(* Schneider Machine Expert - Basic project control_2, file version 2.9.0.0 *)
(* ProjectInformations: Name=Nuevo proyecto *)

HARDWARE
  Cpu 0: TM221M16R/G
  EthernetConfiguration: NetworkName=M221, IpAllocationMode=FixedAddress, IpAddress=0.0.0.0, SubnetMask=0.0.0.0
  SerialLineConfiguration: Baud=Baud19200, Parity=ParityEven, DataBits=DataBits8, StopBits=StopBits1, PhysicalMedium=PhysicalMediumRs485, TransmissionMode=TransmissionModeModbusRtu, SlaveId=1, Addressing=SlaveAddressing
  MastTask: UsePeriodScanMode=true, PeriodScan=50
  FastTask: Period=255
  CpuBehavior: StartingMode=StartAsPreviousState, AutoSaveRamOnEeprom=true, WatchdogPeriod=250

SYMBOLS  (address, symbol, comment, settings)
  %MW271    CONT
  %MW500    ERR
  %MW501    VEL
  %MW502    THETA
  %MW503    CRISP
  %MF1      REAL_ERROR
  %MF10     ENL
  %MF19     ENM
  %MF28     ENP
  %MF37     EZ
  %MF46     EPP
  %MF55     EPM
  %MF64     EPL
  %MF67     REAL_VEL
  %MF76     VNL
  %MF85     VNM
  %MF94     VNP
  %MF103    VZ
  %MF112    VPP
  %MF121    VPM
  %MF130    VPL
  %MF133    REAL_THETA
  %MF142    NL
  %MF151    NM
  %MF160    Z
  %MF169    PM
  %MF178    PL
  %MF181    W1
  %MF184    W2
  %MF187    W3
  %MF190    W4
  %MF193    W5
  %MF196    W6
  %MF199    W7
  %MF202    W8
  %MF205    W9
  %MF208    W10
  %MF211    W11
  %MF214    W12
  %MF217    W13
  %MF220    W14
  %MF223    W15
  %MF226    W16
  %MF229    W17
  %MF232    W18
  %MF235    W19
  %MF238    W20
  %MF241    W21
  %MF244    W22
  %MF247    W23
  %MF250    W24
  %MF253    W25
  %MF256    U_NL
  %MF259    U_NM
  %MF262    U_ZR
  %MF265    U_PM
  %MF268    U_PL
  %KF1      F_CONV  [Value=1000]
  %KF4      CONV_OUTPUT  [Value=100]

POU Nuevo POU
  (* SectionNumber=1 *)

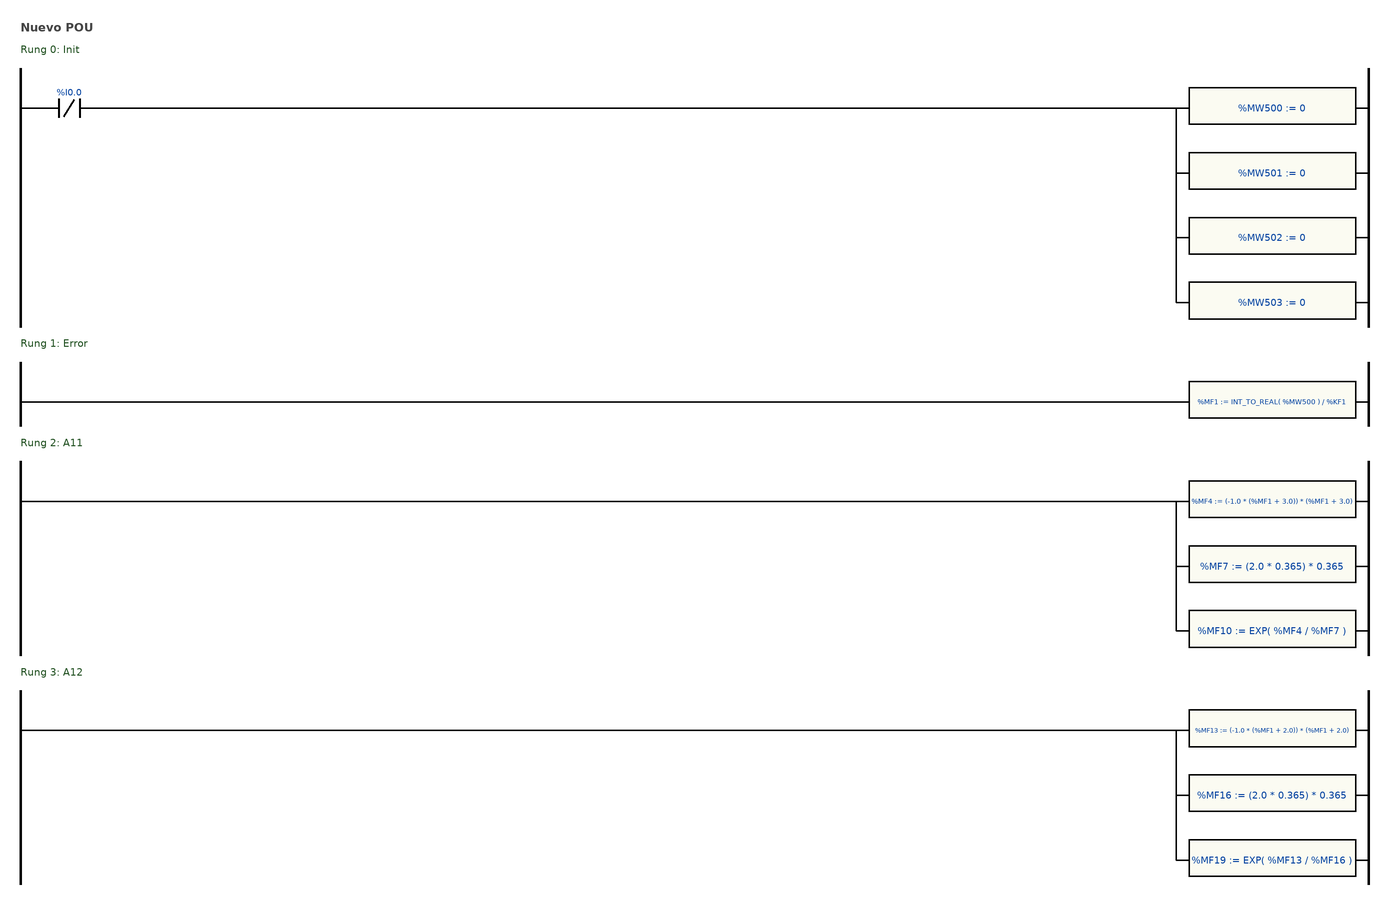

// Rung 0: Init
  LDN %I0.0
  [ %MW500 := 0 ]         (* ERR *)
  [ %MW501 := 0 ]         (* VEL *)
  [ %MW502 := 0 ]         (* THETA *)
  [ %MW503 := 0 ]         (* CRISP *)
  // as ST:
  //   IF NOT %I0.0 THEN ERR := 0; END_IF;
  //   IF NOT %I0.0 THEN VEL := 0; END_IF;
  //   IF NOT %I0.0 THEN THETA := 0; END_IF;
  //   IF NOT %I0.0 THEN CRISP := 0; END_IF;

// Rung 1: Error
  LD 1
  [ %MF1 := INT_TO_REAL ( %MW500 ) / %KF1 ](* REAL_ERROR, ERR, F_CONV *)
  // as ST:
  //   REAL_ERROR := INT_TO_REAL ( ERR ) / F_CONV;

// Rung 2: A11
  LD 1
  [ %MF4 := ( -1.0 * ( %MF1 + 3.0 ) ) * ( %MF1 + 3.0 ) ](* REAL_ERROR, REAL_ERROR *)
  [ %MF7 := ( 2.0 * 0.365 ) * 0.365 ]
  [ %MF10 := EXP ( %MF4 / %MF7 ) ](* ENL *)
  // as ST:
  //   %MF4 := ( -1.0 * ( REAL_ERROR + 3.0 ) ) * ( REAL_ERROR + 3.0 );
  //   %MF7 := ( 2.0 * 0.365 ) * 0.365;
  //   ENL := EXP ( %MF4 / %MF7 );

// Rung 3: A12
  LD 1
  [ %MF13 := ( -1.0 * ( %MF1 + 2.0 ) ) * ( %MF1 + 2.0 ) ](* REAL_ERROR, REAL_ERROR *)
  [ %MF16 := ( 2.0 * 0.365 ) * 0.365 ]
  [ %MF19 := EXP ( %MF13 / %MF16 ) ](* ENM *)
  // as ST:
  //   %MF13 := ( -1.0 * ( REAL_ERROR + 2.0 ) ) * ( REAL_ERROR + 2.0 );
  //   %MF16 := ( 2.0 * 0.365 ) * 0.365;
  //   ENM := EXP ( %MF13 / %MF16 );

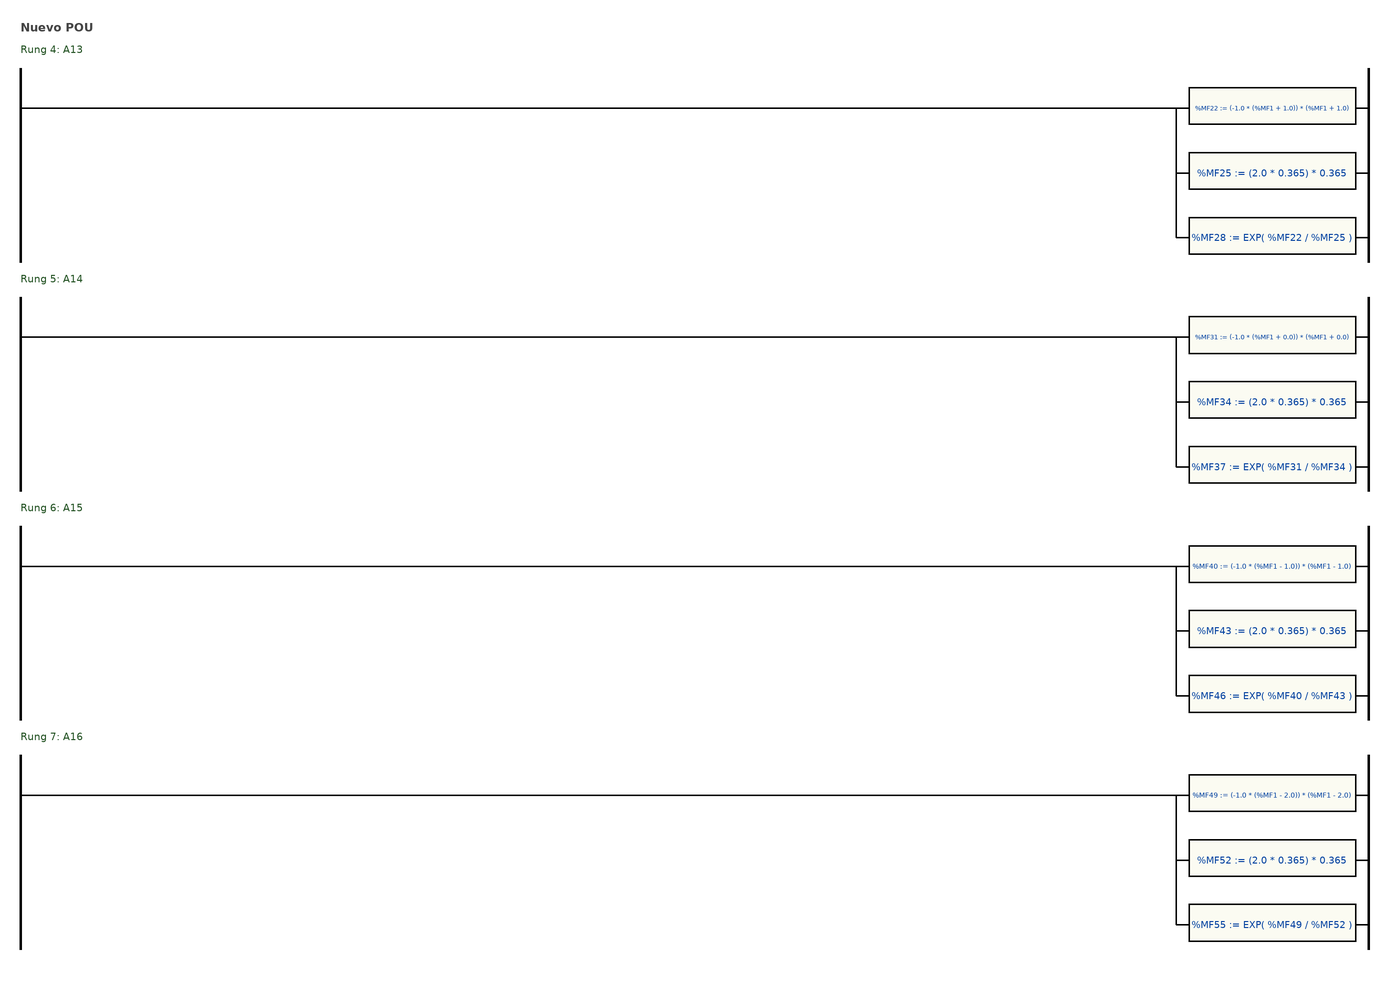

// Rung 4: A13
  LD 1
  [ %MF22 := ( -1.0 * ( %MF1 + 1.0 ) ) * ( %MF1 + 1.0 ) ](* REAL_ERROR, REAL_ERROR *)
  [ %MF25 := ( 2.0 * 0.365 ) * 0.365 ]
  [ %MF28 := EXP ( %MF22 / %MF25 ) ](* ENP *)
  // as ST:
  //   %MF22 := ( -1.0 * ( REAL_ERROR + 1.0 ) ) * ( REAL_ERROR + 1.0 );
  //   %MF25 := ( 2.0 * 0.365 ) * 0.365;
  //   ENP := EXP ( %MF22 / %MF25 );

// Rung 5: A14
  LD 1
  [ %MF31 := ( -1.0 * ( %MF1 + 0.0 ) ) * ( %MF1 + 0.0 ) ](* REAL_ERROR, REAL_ERROR *)
  [ %MF34 := ( 2.0 * 0.365 ) * 0.365 ]
  [ %MF37 := EXP ( %MF31 / %MF34 ) ](* EZ *)
  // as ST:
  //   %MF31 := ( -1.0 * ( REAL_ERROR + 0.0 ) ) * ( REAL_ERROR + 0.0 );
  //   %MF34 := ( 2.0 * 0.365 ) * 0.365;
  //   EZ := EXP ( %MF31 / %MF34 );

// Rung 6: A15
  LD 1
  [ %MF40 := ( -1.0 * ( %MF1 - 1.0 ) ) * ( %MF1 - 1.0 ) ](* REAL_ERROR, REAL_ERROR *)
  [ %MF43 := ( 2.0 * 0.365 ) * 0.365 ]
  [ %MF46 := EXP ( %MF40 / %MF43 ) ](* EPP *)
  // as ST:
  //   %MF40 := ( -1.0 * ( REAL_ERROR - 1.0 ) ) * ( REAL_ERROR - 1.0 );
  //   %MF43 := ( 2.0 * 0.365 ) * 0.365;
  //   EPP := EXP ( %MF40 / %MF43 );

// Rung 7: A16
  LD 1
  [ %MF49 := ( -1.0 * ( %MF1 - 2.0 ) ) * ( %MF1 - 2.0 ) ](* REAL_ERROR, REAL_ERROR *)
  [ %MF52 := ( 2.0 * 0.365 ) * 0.365 ]
  [ %MF55 := EXP ( %MF49 / %MF52 ) ](* EPM *)
  // as ST:
  //   %MF49 := ( -1.0 * ( REAL_ERROR - 2.0 ) ) * ( REAL_ERROR - 2.0 );
  //   %MF52 := ( 2.0 * 0.365 ) * 0.365;
  //   EPM := EXP ( %MF49 / %MF52 );

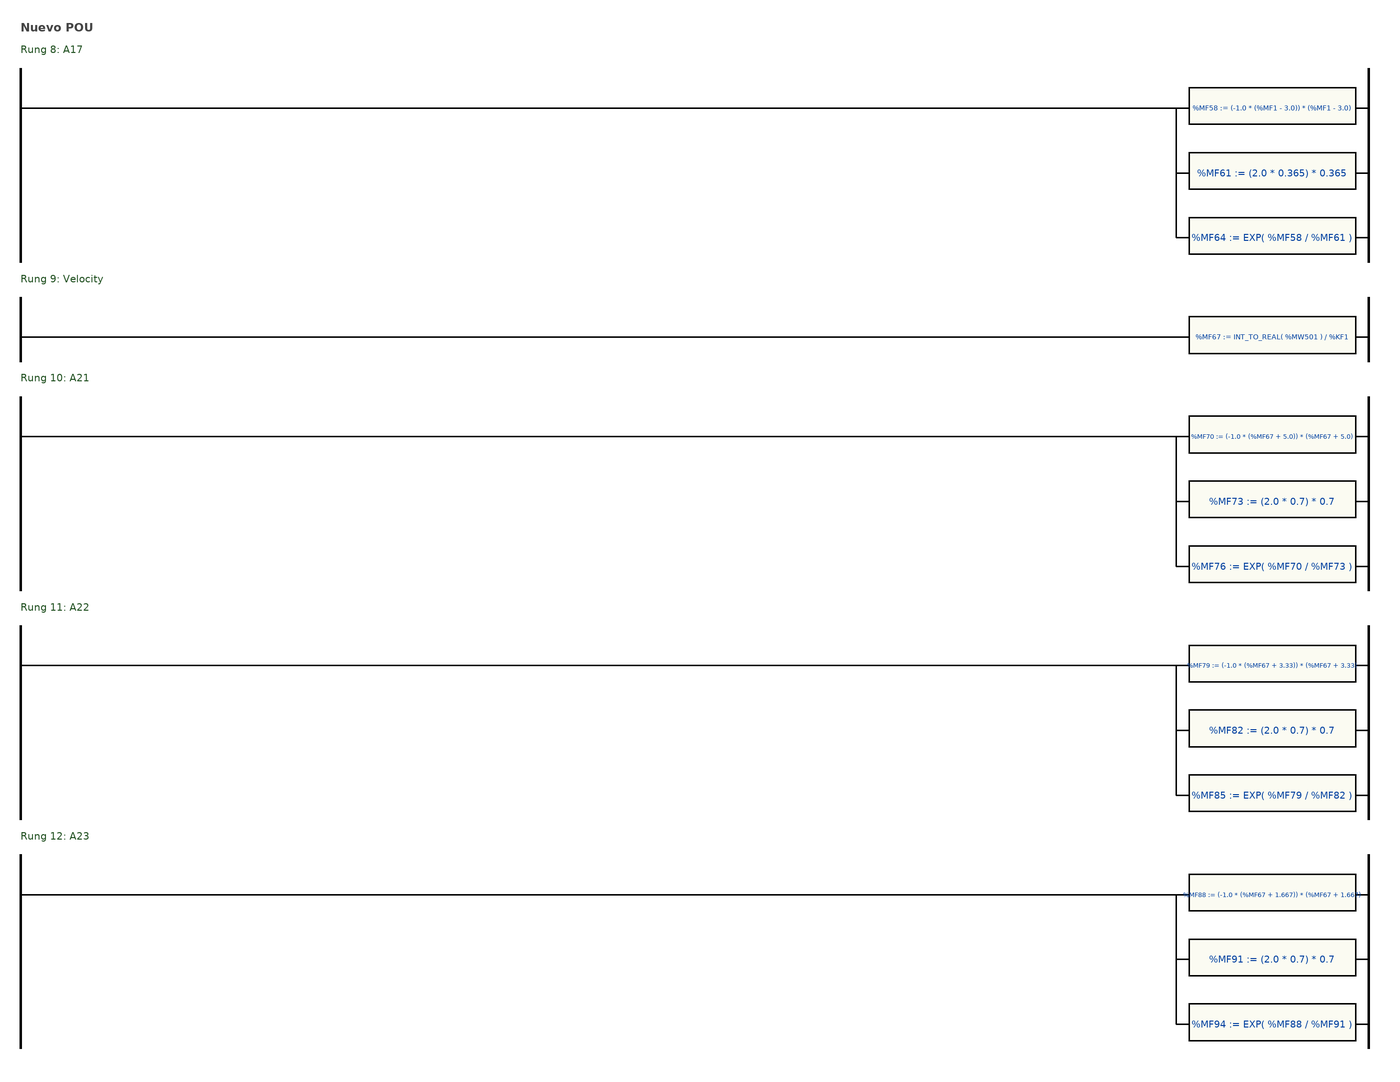

// Rung 8: A17
  LD 1
  [ %MF58 := ( -1.0 * ( %MF1 - 3.0 ) ) * ( %MF1 - 3.0 ) ](* REAL_ERROR, REAL_ERROR *)
  [ %MF61 := ( 2.0 * 0.365 ) * 0.365 ]
  [ %MF64 := EXP ( %MF58 / %MF61 ) ](* EPL *)
  // as ST:
  //   %MF58 := ( -1.0 * ( REAL_ERROR - 3.0 ) ) * ( REAL_ERROR - 3.0 );
  //   %MF61 := ( 2.0 * 0.365 ) * 0.365;
  //   EPL := EXP ( %MF58 / %MF61 );

// Rung 9: Velocity
  LD 1
  [ %MF67 := INT_TO_REAL ( %MW501 ) / %KF1 ](* REAL_VEL, VEL, F_CONV *)
  // as ST:
  //   REAL_VEL := INT_TO_REAL ( VEL ) / F_CONV;

// Rung 10: A21
  LD 1
  [ %MF70 := ( -1.0 * ( %MF67 + 5.0 ) ) * ( %MF67 + 5.0 ) ](* REAL_VEL, REAL_VEL *)
  [ %MF73 := ( 2.0 * 0.7 ) * 0.7 ]
  [ %MF76 := EXP ( %MF70 / %MF73 ) ](* VNL *)
  // as ST:
  //   %MF70 := ( -1.0 * ( REAL_VEL + 5.0 ) ) * ( REAL_VEL + 5.0 );
  //   %MF73 := ( 2.0 * 0.7 ) * 0.7;
  //   VNL := EXP ( %MF70 / %MF73 );

// Rung 11: A22
  LD 1
  [ %MF79 := ( -1.0 * ( %MF67 + 3.33 ) ) * ( %MF67 + 3.33 ) ](* REAL_VEL, REAL_VEL *)
  [ %MF82 := ( 2.0 * 0.7 ) * 0.7 ]
  [ %MF85 := EXP ( %MF79 / %MF82 ) ](* VNM *)
  // as ST:
  //   %MF79 := ( -1.0 * ( REAL_VEL + 3.33 ) ) * ( REAL_VEL + 3.33 );
  //   %MF82 := ( 2.0 * 0.7 ) * 0.7;
  //   VNM := EXP ( %MF79 / %MF82 );

// Rung 12: A23
  LD 1
  [ %MF88 := ( -1.0 * ( %MF67 + 1.667 ) ) * ( %MF67 + 1.667 ) ](* REAL_VEL, REAL_VEL *)
  [ %MF91 := ( 2.0 * 0.7 ) * 0.7 ]
  [ %MF94 := EXP ( %MF88 / %MF91 ) ](* VNP *)
  // as ST:
  //   %MF88 := ( -1.0 * ( REAL_VEL + 1.667 ) ) * ( REAL_VEL + 1.667 );
  //   %MF91 := ( 2.0 * 0.7 ) * 0.7;
  //   VNP := EXP ( %MF88 / %MF91 );

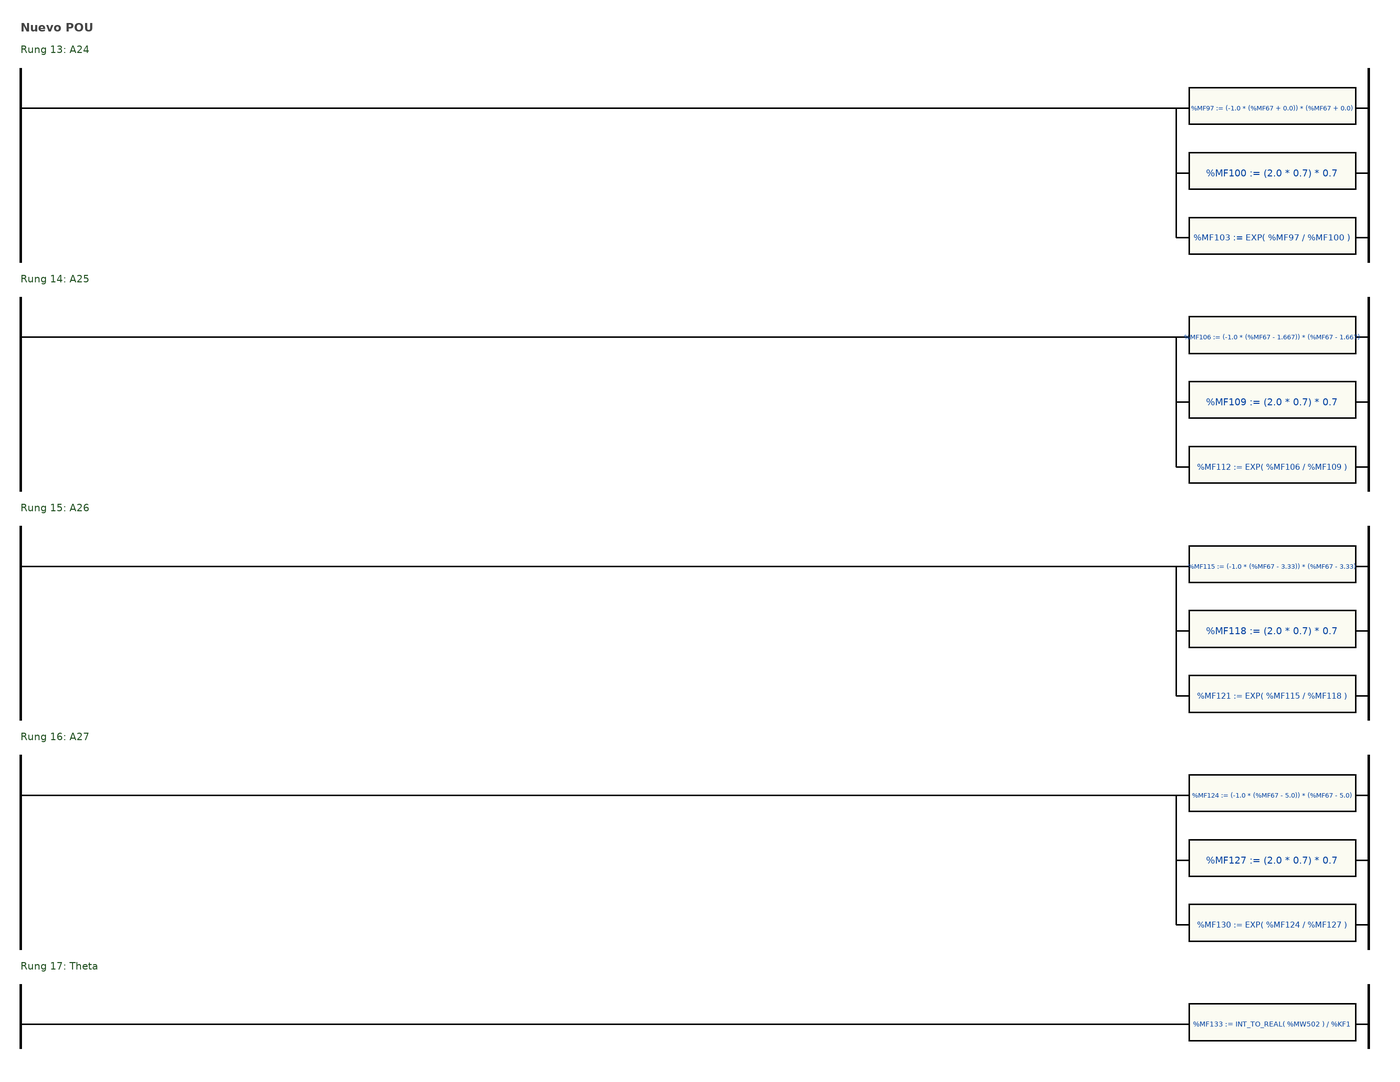

// Rung 13: A24
  LD 1
  [ %MF97 := ( -1.0 * ( %MF67 + 0.0 ) ) * ( %MF67 + 0.0 ) ](* REAL_VEL, REAL_VEL *)
  [ %MF100 := ( 2.0 * 0.7 ) * 0.7 ]
  [ %MF103 := EXP ( %MF97 / %MF100 ) ](* VZ *)
  // as ST:
  //   %MF97 := ( -1.0 * ( REAL_VEL + 0.0 ) ) * ( REAL_VEL + 0.0 );
  //   %MF100 := ( 2.0 * 0.7 ) * 0.7;
  //   VZ := EXP ( %MF97 / %MF100 );

// Rung 14: A25
  LD 1
  [ %MF106 := ( -1.0 * ( %MF67 - 1.667 ) ) * ( %MF67 - 1.667 ) ](* REAL_VEL, REAL_VEL *)
  [ %MF109 := ( 2.0 * 0.7 ) * 0.7 ]
  [ %MF112 := EXP ( %MF106 / %MF109 ) ](* VPP *)
  // as ST:
  //   %MF106 := ( -1.0 * ( REAL_VEL - 1.667 ) ) * ( REAL_VEL - 1.667 );
  //   %MF109 := ( 2.0 * 0.7 ) * 0.7;
  //   VPP := EXP ( %MF106 / %MF109 );

// Rung 15: A26
  LD 1
  [ %MF115 := ( -1.0 * ( %MF67 - 3.33 ) ) * ( %MF67 - 3.33 ) ](* REAL_VEL, REAL_VEL *)
  [ %MF118 := ( 2.0 * 0.7 ) * 0.7 ]
  [ %MF121 := EXP ( %MF115 / %MF118 ) ](* VPM *)
  // as ST:
  //   %MF115 := ( -1.0 * ( REAL_VEL - 3.33 ) ) * ( REAL_VEL - 3.33 );
  //   %MF118 := ( 2.0 * 0.7 ) * 0.7;
  //   VPM := EXP ( %MF115 / %MF118 );

// Rung 16: A27
  LD 1
  [ %MF124 := ( -1.0 * ( %MF67 - 5.0 ) ) * ( %MF67 - 5.0 ) ](* REAL_VEL, REAL_VEL *)
  [ %MF127 := ( 2.0 * 0.7 ) * 0.7 ]
  [ %MF130 := EXP ( %MF124 / %MF127 ) ](* VPL *)
  // as ST:
  //   %MF124 := ( -1.0 * ( REAL_VEL - 5.0 ) ) * ( REAL_VEL - 5.0 );
  //   %MF127 := ( 2.0 * 0.7 ) * 0.7;
  //   VPL := EXP ( %MF124 / %MF127 );

// Rung 17: Theta
  LD 1
  [ %MF133 := INT_TO_REAL ( %MW502 ) / %KF1 ](* REAL_THETA, THETA, F_CONV *)
  // as ST:
  //   REAL_THETA := INT_TO_REAL ( THETA ) / F_CONV;

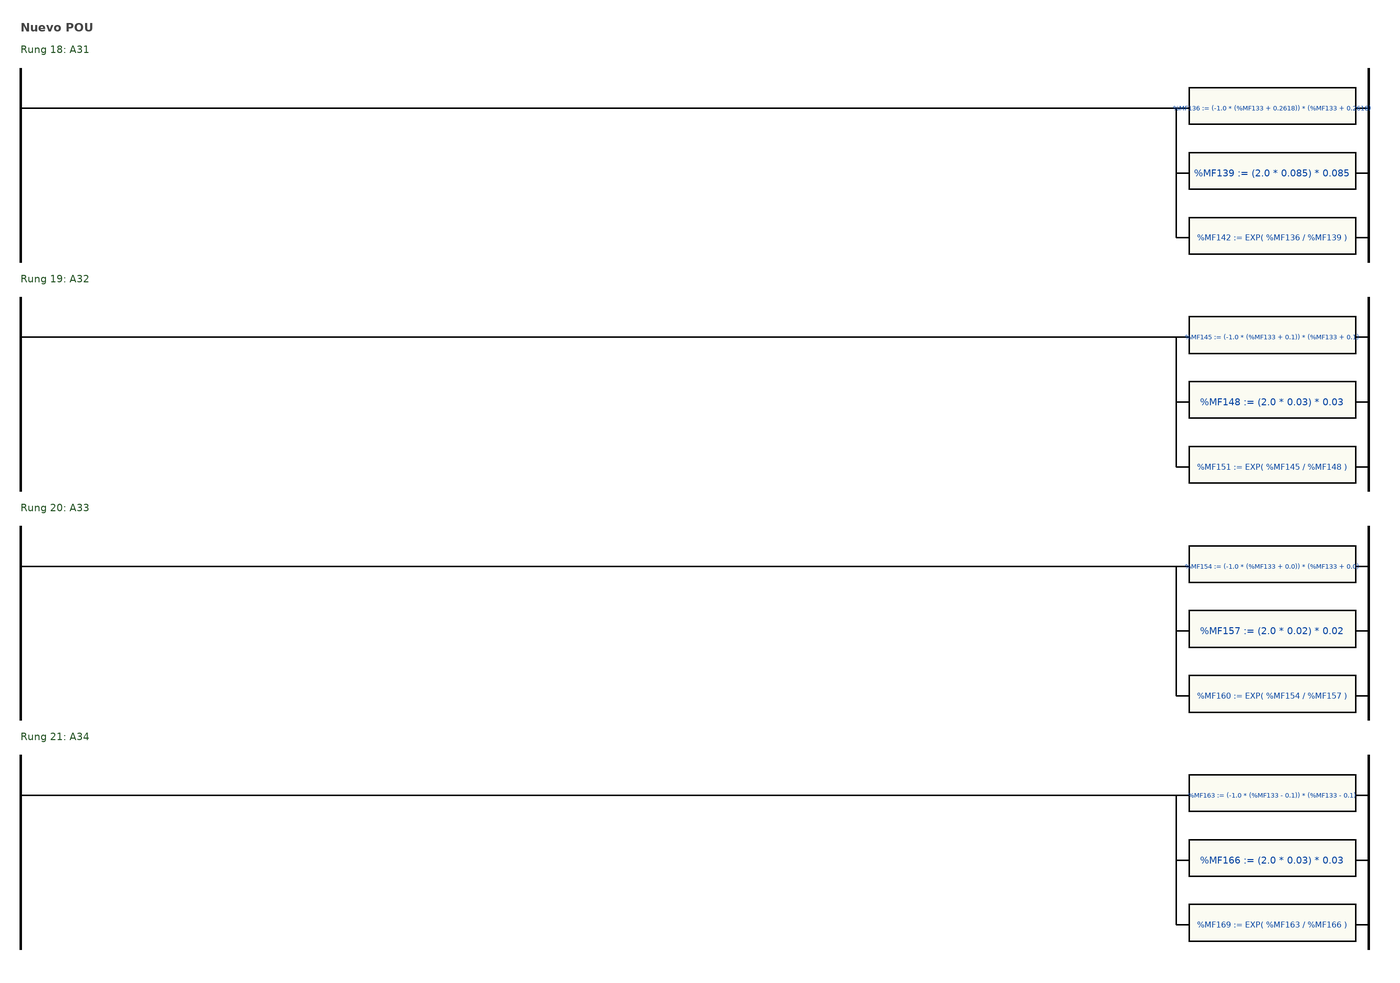

// Rung 18: A31
  LD 1
  [ %MF136 := ( -1.0 * ( %MF133 + 0.2618 ) ) * ( %MF133 + 0.2618 ) ](* REAL_THETA, REAL_THETA *)
  [ %MF139 := ( 2.0 * 0.085 ) * 0.085 ]
  [ %MF142 := EXP ( %MF136 / %MF139 ) ](* NL *)
  // as ST:
  //   %MF136 := ( -1.0 * ( REAL_THETA + 0.2618 ) ) * ( REAL_THETA + 0.2618 );
  //   %MF139 := ( 2.0 * 0.085 ) * 0.085;
  //   NL := EXP ( %MF136 / %MF139 );

// Rung 19: A32
  LD 1
  [ %MF145 := ( -1.0 * ( %MF133 + 0.1 ) ) * ( %MF133 + 0.1 ) ](* REAL_THETA, REAL_THETA *)
  [ %MF148 := ( 2.0 * 0.03 ) * 0.03 ]
  [ %MF151 := EXP ( %MF145 / %MF148 ) ](* NM *)
  // as ST:
  //   %MF145 := ( -1.0 * ( REAL_THETA + 0.1 ) ) * ( REAL_THETA + 0.1 );
  //   %MF148 := ( 2.0 * 0.03 ) * 0.03;
  //   NM := EXP ( %MF145 / %MF148 );

// Rung 20: A33
  LD 1
  [ %MF154 := ( -1.0 * ( %MF133 + 0.0 ) ) * ( %MF133 + 0.0 ) ](* REAL_THETA, REAL_THETA *)
  [ %MF157 := ( 2.0 * 0.02 ) * 0.02 ]
  [ %MF160 := EXP ( %MF154 / %MF157 ) ](* Z *)
  // as ST:
  //   %MF154 := ( -1.0 * ( REAL_THETA + 0.0 ) ) * ( REAL_THETA + 0.0 );
  //   %MF157 := ( 2.0 * 0.02 ) * 0.02;
  //   Z := EXP ( %MF154 / %MF157 );

// Rung 21: A34
  LD 1
  [ %MF163 := ( -1.0 * ( %MF133 - 0.1 ) ) * ( %MF133 - 0.1 ) ](* REAL_THETA, REAL_THETA *)
  [ %MF166 := ( 2.0 * 0.03 ) * 0.03 ]
  [ %MF169 := EXP ( %MF163 / %MF166 ) ](* PM *)
  // as ST:
  //   %MF163 := ( -1.0 * ( REAL_THETA - 0.1 ) ) * ( REAL_THETA - 0.1 );
  //   %MF166 := ( 2.0 * 0.03 ) * 0.03;
  //   PM := EXP ( %MF163 / %MF166 );

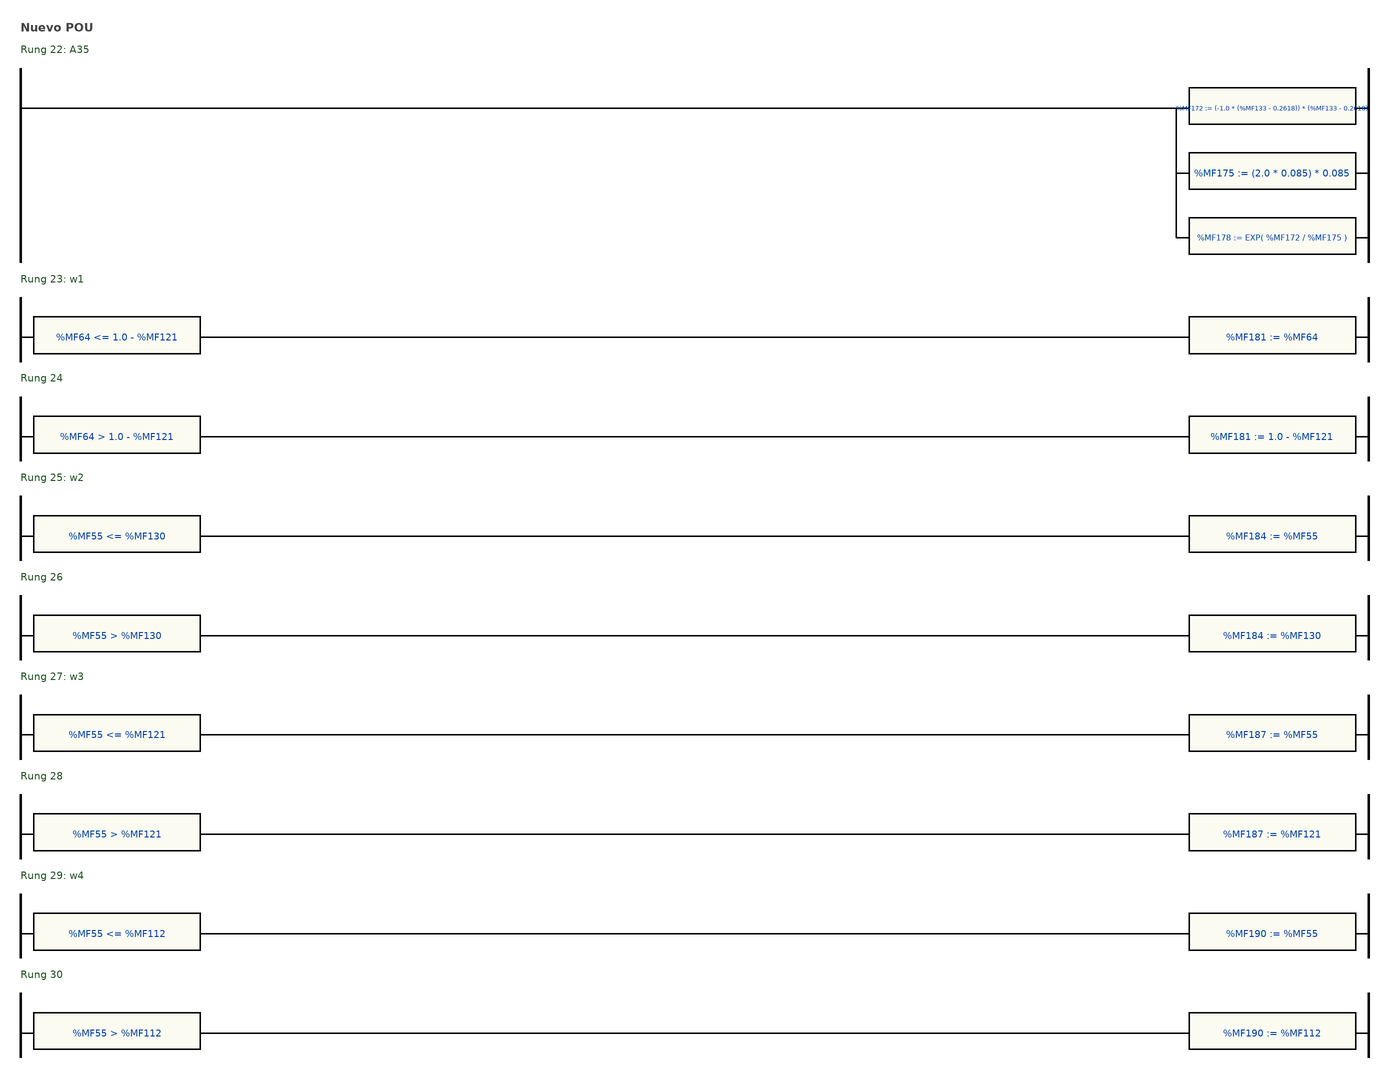

// Rung 22: A35
  LD 1
  [ %MF172 := ( -1.0 * ( %MF133 - 0.2618 ) ) * ( %MF133 - 0.2618 ) ](* REAL_THETA, REAL_THETA *)
  [ %MF175 := ( 2.0 * 0.085 ) * 0.085 ]
  [ %MF178 := EXP ( %MF172 / %MF175 ) ](* PL *)
  // as ST:
  //   %MF172 := ( -1.0 * ( REAL_THETA - 0.2618 ) ) * ( REAL_THETA - 0.2618 );
  //   %MF175 := ( 2.0 * 0.085 ) * 0.085;
  //   PL := EXP ( %MF172 / %MF175 );

// Rung 23: w1
  LD 1
  AND [ %MF64 <= 1.0 - %MF121 ](* EPL, VPM *)
  [ %MF181 := %MF64 ]     (* W1, EPL *)
  // as ST:
  //   IF EPL <= 1.0 - VPM THEN W1 := EPL; END_IF;

// Rung 24
  LD 1
  AND [ %MF64 > 1.0 - %MF121 ](* EPL, VPM *)
  [ %MF181 := 1.0 - %MF121 ](* W1, VPM *)
  // as ST:
  //   IF EPL > 1.0 - VPM THEN W1 := 1.0 - VPM; END_IF;

// Rung 25: w2
  LD [ %MF55 <= %MF130 ]  (* EPM, VPL *)
  [ %MF184 := %MF55 ]     (* W2, EPM *)
  // as ST:
  //   IF EPM <= VPL THEN W2 := EPM; END_IF;

// Rung 26
  LD [ %MF55 > %MF130 ]   (* EPM, VPL *)
  [ %MF184 := %MF130 ]    (* W2, VPL *)
  // as ST:
  //   IF EPM > VPL THEN W2 := VPL; END_IF;

// Rung 27: w3
  LD [ %MF55 <= %MF121 ]  (* EPM, VPM *)
  [ %MF187 := %MF55 ]     (* W3, EPM *)
  // as ST:
  //   IF EPM <= VPM THEN W3 := EPM; END_IF;

// Rung 28
  LD [ %MF55 > %MF121 ]   (* EPM, VPM *)
  [ %MF187 := %MF121 ]    (* W3, VPM *)
  // as ST:
  //   IF EPM > VPM THEN W3 := VPM; END_IF;

// Rung 29: w4
  LD [ %MF55 <= %MF112 ]  (* EPM, VPP *)
  [ %MF190 := %MF55 ]     (* W4, EPM *)
  // as ST:
  //   IF EPM <= VPP THEN W4 := EPM; END_IF;

// Rung 30
  LD [ %MF55 > %MF112 ]   (* EPM, VPP *)
  [ %MF190 := %MF112 ]    (* W4, VPP *)
  // as ST:
  //   IF EPM > VPP THEN W4 := VPP; END_IF;

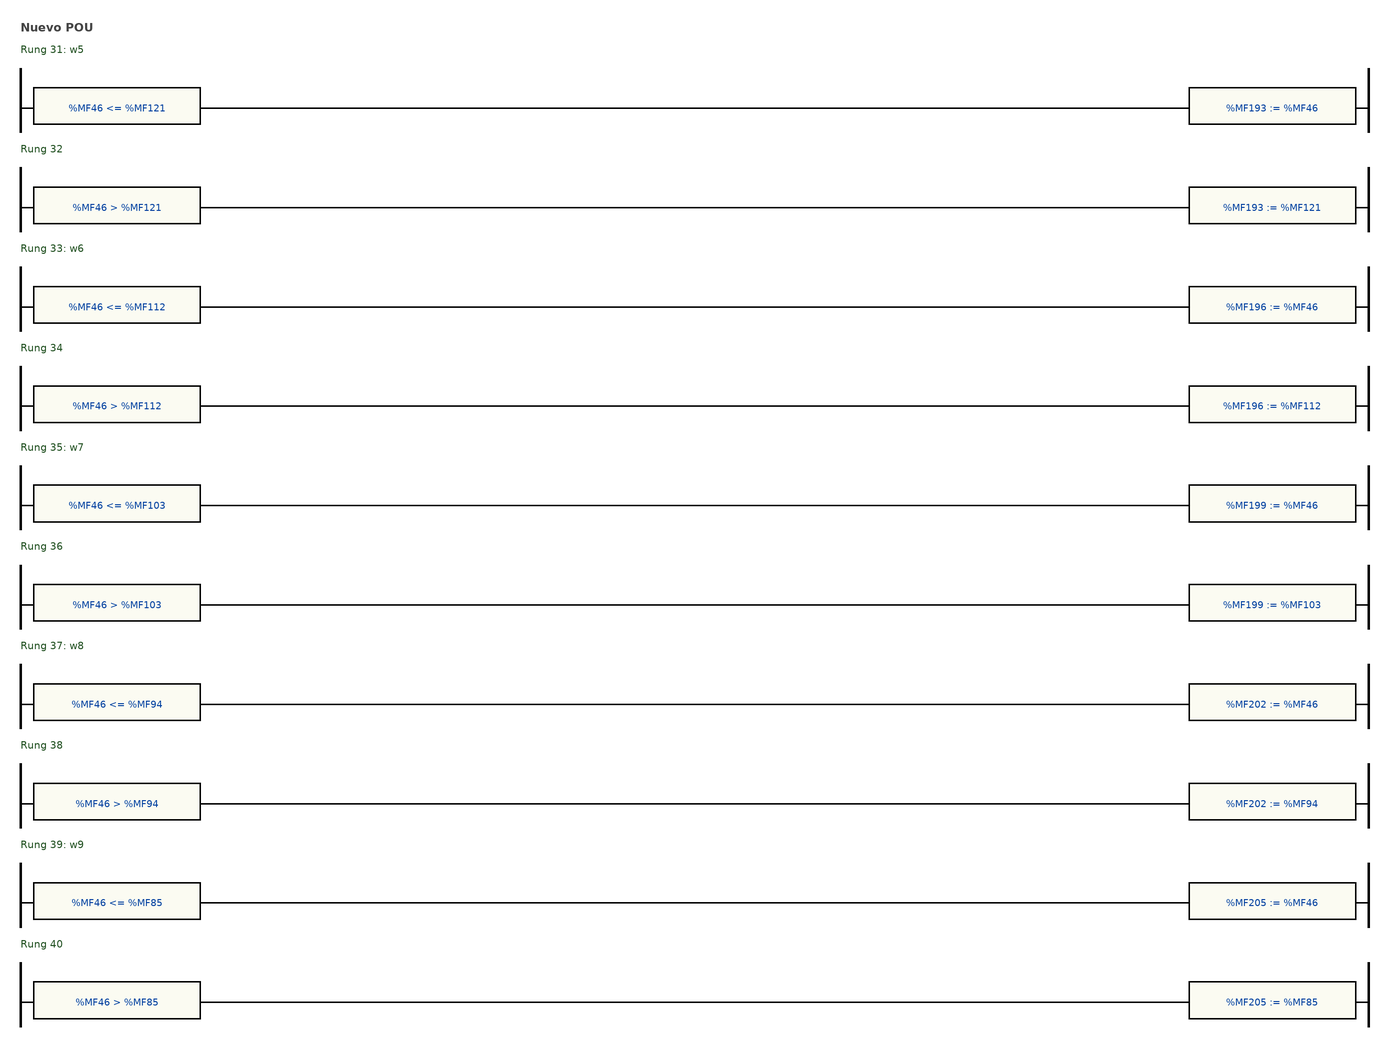

// Rung 31: w5
  LD [ %MF46 <= %MF121 ]  (* EPP, VPM *)
  [ %MF193 := %MF46 ]     (* W5, EPP *)
  // as ST:
  //   IF EPP <= VPM THEN W5 := EPP; END_IF;

// Rung 32
  LD [ %MF46 > %MF121 ]   (* EPP, VPM *)
  [ %MF193 := %MF121 ]    (* W5, VPM *)
  // as ST:
  //   IF EPP > VPM THEN W5 := VPM; END_IF;

// Rung 33: w6
  LD [ %MF46 <= %MF112 ]  (* EPP, VPP *)
  [ %MF196 := %MF46 ]     (* W6, EPP *)
  // as ST:
  //   IF EPP <= VPP THEN W6 := EPP; END_IF;

// Rung 34
  LD [ %MF46 > %MF112 ]   (* EPP, VPP *)
  [ %MF196 := %MF112 ]    (* W6, VPP *)
  // as ST:
  //   IF EPP > VPP THEN W6 := VPP; END_IF;

// Rung 35: w7
  LD [ %MF46 <= %MF103 ]  (* EPP, VZ *)
  [ %MF199 := %MF46 ]     (* W7, EPP *)
  // as ST:
  //   IF EPP <= VZ THEN W7 := EPP; END_IF;

// Rung 36
  LD [ %MF46 > %MF103 ]   (* EPP, VZ *)
  [ %MF199 := %MF103 ]    (* W7, VZ *)
  // as ST:
  //   IF EPP > VZ THEN W7 := VZ; END_IF;

// Rung 37: w8
  LD [ %MF46 <= %MF94 ]   (* EPP, VNP *)
  [ %MF202 := %MF46 ]     (* W8, EPP *)
  // as ST:
  //   IF EPP <= VNP THEN W8 := EPP; END_IF;

// Rung 38
  LD [ %MF46 > %MF94 ]    (* EPP, VNP *)
  [ %MF202 := %MF94 ]     (* W8, VNP *)
  // as ST:
  //   IF EPP > VNP THEN W8 := VNP; END_IF;

// Rung 39: w9
  LD [ %MF46 <= %MF85 ]   (* EPP, VNM *)
  [ %MF205 := %MF46 ]     (* W9, EPP *)
  // as ST:
  //   IF EPP <= VNM THEN W9 := EPP; END_IF;

// Rung 40
  LD [ %MF46 > %MF85 ]    (* EPP, VNM *)
  [ %MF205 := %MF85 ]     (* W9, VNM *)
  // as ST:
  //   IF EPP > VNM THEN W9 := VNM; END_IF;

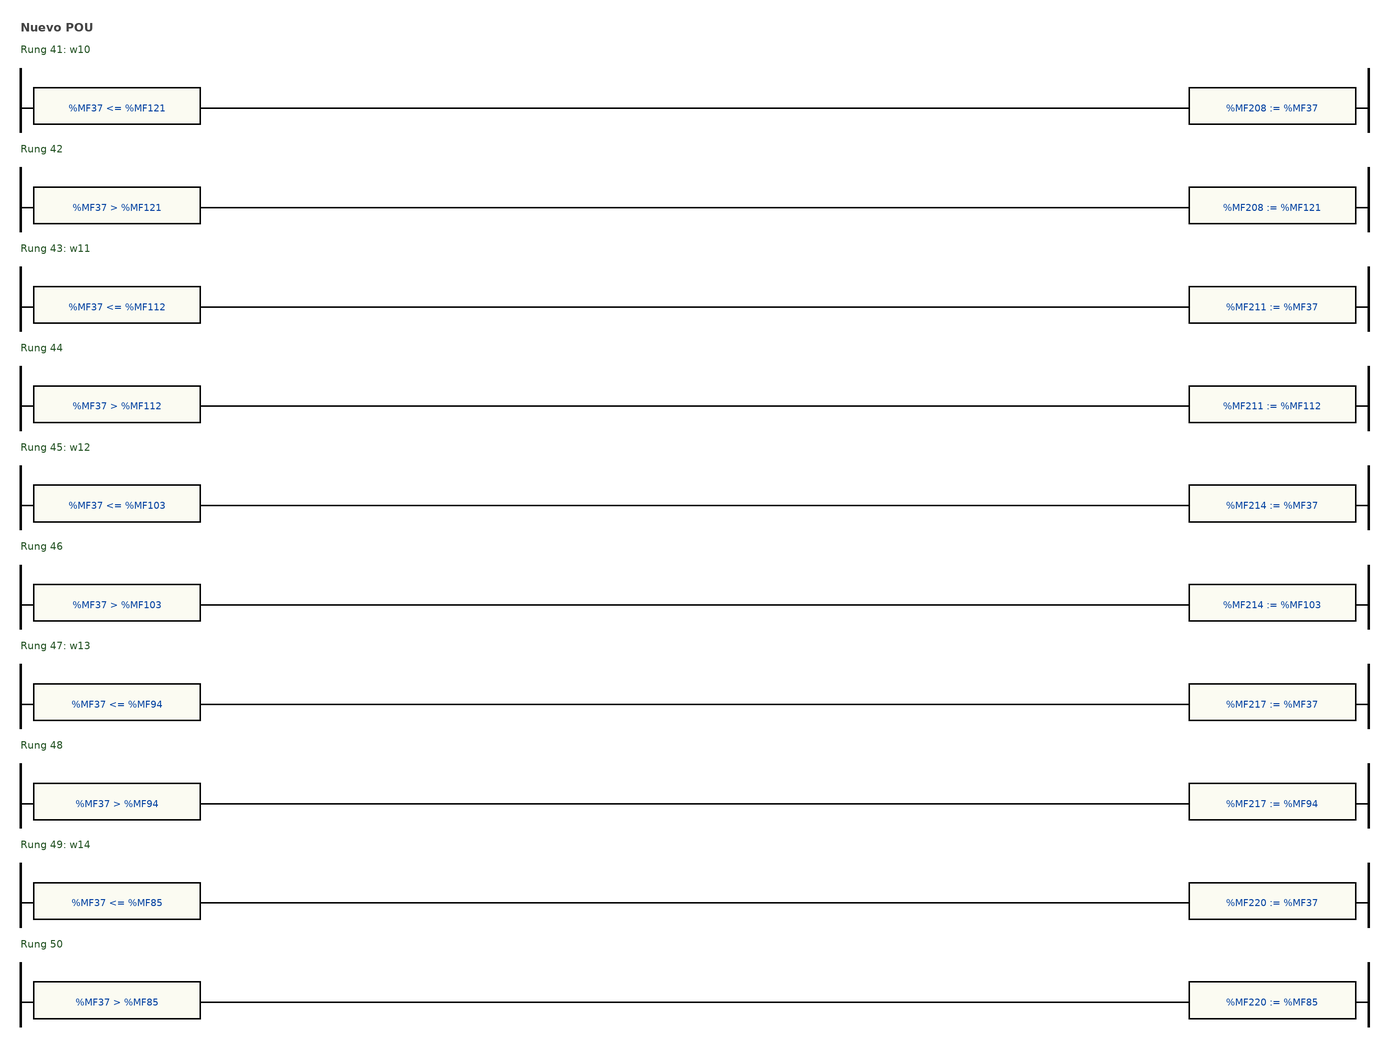

// Rung 41: w10
  LD [ %MF37 <= %MF121 ]  (* EZ, VPM *)
  [ %MF208 := %MF37 ]     (* W10, EZ *)
  // as ST:
  //   IF EZ <= VPM THEN W10 := EZ; END_IF;

// Rung 42
  LD [ %MF37 > %MF121 ]   (* EZ, VPM *)
  [ %MF208 := %MF121 ]    (* W10, VPM *)
  // as ST:
  //   IF EZ > VPM THEN W10 := VPM; END_IF;

// Rung 43: w11
  LD [ %MF37 <= %MF112 ]  (* EZ, VPP *)
  [ %MF211 := %MF37 ]     (* W11, EZ *)
  // as ST:
  //   IF EZ <= VPP THEN W11 := EZ; END_IF;

// Rung 44
  LD [ %MF37 > %MF112 ]   (* EZ, VPP *)
  [ %MF211 := %MF112 ]    (* W11, VPP *)
  // as ST:
  //   IF EZ > VPP THEN W11 := VPP; END_IF;

// Rung 45: w12
  LD [ %MF37 <= %MF103 ]  (* EZ, VZ *)
  [ %MF214 := %MF37 ]     (* W12, EZ *)
  // as ST:
  //   IF EZ <= VZ THEN W12 := EZ; END_IF;

// Rung 46
  LD [ %MF37 > %MF103 ]   (* EZ, VZ *)
  [ %MF214 := %MF103 ]    (* W12, VZ *)
  // as ST:
  //   IF EZ > VZ THEN W12 := VZ; END_IF;

// Rung 47: w13
  LD [ %MF37 <= %MF94 ]   (* EZ, VNP *)
  [ %MF217 := %MF37 ]     (* W13, EZ *)
  // as ST:
  //   IF EZ <= VNP THEN W13 := EZ; END_IF;

// Rung 48
  LD [ %MF37 > %MF94 ]    (* EZ, VNP *)
  [ %MF217 := %MF94 ]     (* W13, VNP *)
  // as ST:
  //   IF EZ > VNP THEN W13 := VNP; END_IF;

// Rung 49: w14
  LD [ %MF37 <= %MF85 ]   (* EZ, VNM *)
  [ %MF220 := %MF37 ]     (* W14, EZ *)
  // as ST:
  //   IF EZ <= VNM THEN W14 := EZ; END_IF;

// Rung 50
  LD [ %MF37 > %MF85 ]    (* EZ, VNM *)
  [ %MF220 := %MF85 ]     (* W14, VNM *)
  // as ST:
  //   IF EZ > VNM THEN W14 := VNM; END_IF;

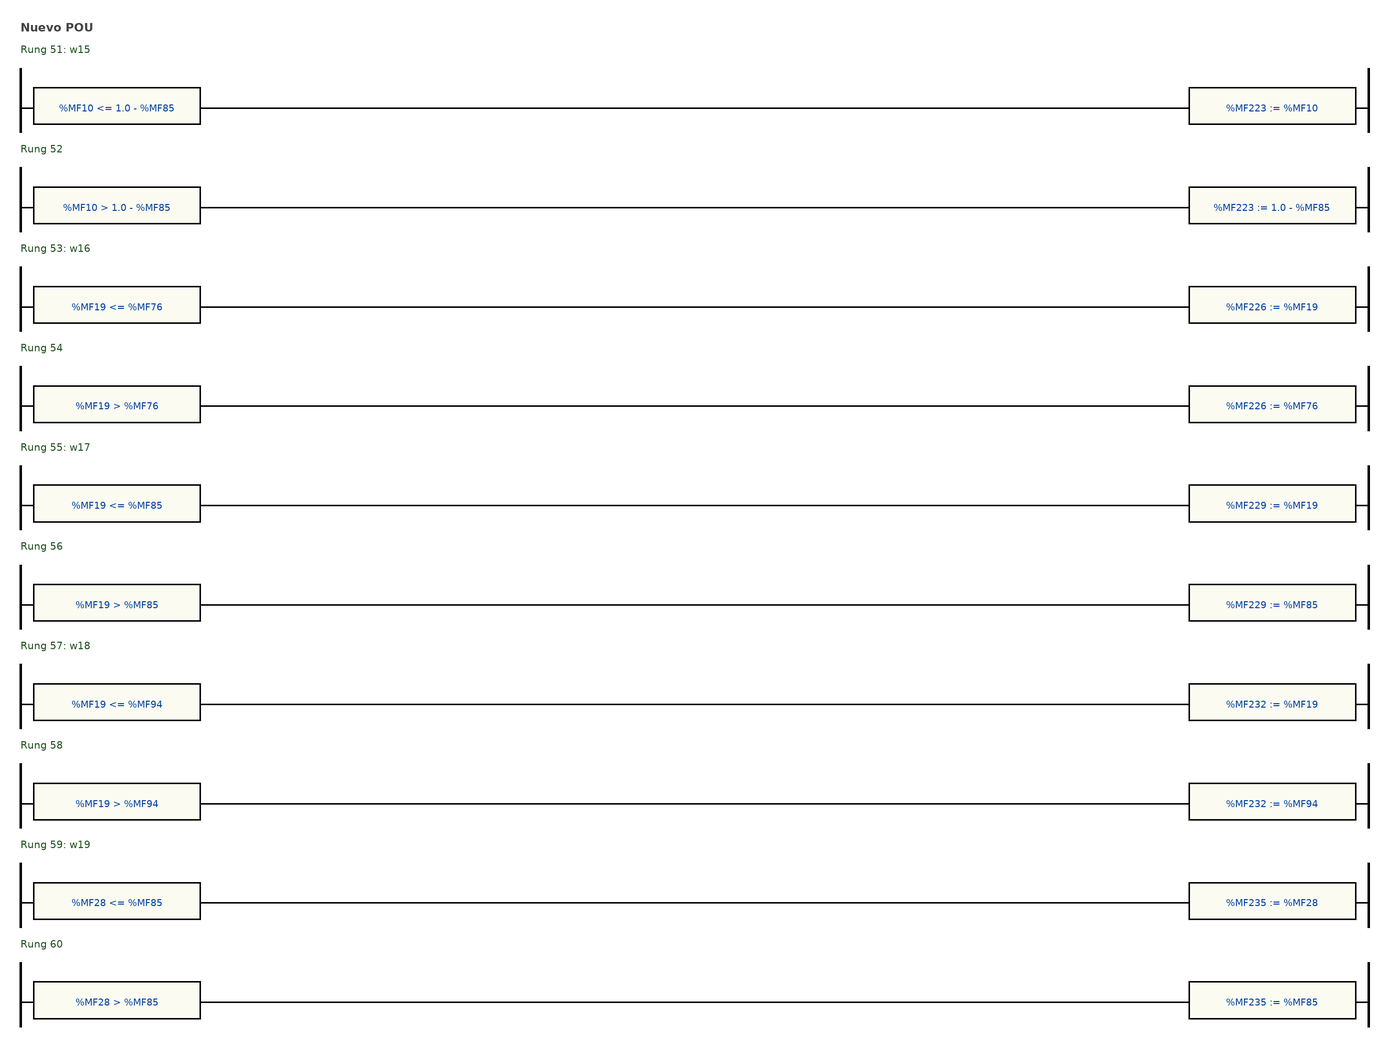

// Rung 51: w15
  LD 1
  AND [ %MF10 <= 1.0 - %MF85 ](* ENL, VNM *)
  [ %MF223 := %MF10 ]     (* W15, ENL *)
  // as ST:
  //   IF ENL <= 1.0 - VNM THEN W15 := ENL; END_IF;

// Rung 52
  LD 1
  AND [ %MF10 > 1.0 - %MF85 ](* ENL, VNM *)
  [ %MF223 := 1.0 - %MF85 ](* W15, VNM *)
  // as ST:
  //   IF ENL > 1.0 - VNM THEN W15 := 1.0 - VNM; END_IF;

// Rung 53: w16
  LD [ %MF19 <= %MF76 ]   (* ENM, VNL *)
  [ %MF226 := %MF19 ]     (* W16, ENM *)
  // as ST:
  //   IF ENM <= VNL THEN W16 := ENM; END_IF;

// Rung 54
  LD [ %MF19 > %MF76 ]    (* ENM, VNL *)
  [ %MF226 := %MF76 ]     (* W16, VNL *)
  // as ST:
  //   IF ENM > VNL THEN W16 := VNL; END_IF;

// Rung 55: w17
  LD [ %MF19 <= %MF85 ]   (* ENM, VNM *)
  [ %MF229 := %MF19 ]     (* W17, ENM *)
  // as ST:
  //   IF ENM <= VNM THEN W17 := ENM; END_IF;

// Rung 56
  LD [ %MF19 > %MF85 ]    (* ENM, VNM *)
  [ %MF229 := %MF85 ]     (* W17, VNM *)
  // as ST:
  //   IF ENM > VNM THEN W17 := VNM; END_IF;

// Rung 57: w18
  LD [ %MF19 <= %MF94 ]   (* ENM, VNP *)
  [ %MF232 := %MF19 ]     (* W18, ENM *)
  // as ST:
  //   IF ENM <= VNP THEN W18 := ENM; END_IF;

// Rung 58
  LD [ %MF19 > %MF94 ]    (* ENM, VNP *)
  [ %MF232 := %MF94 ]     (* W18, VNP *)
  // as ST:
  //   IF ENM > VNP THEN W18 := VNP; END_IF;

// Rung 59: w19
  LD [ %MF28 <= %MF85 ]   (* ENP, VNM *)
  [ %MF235 := %MF28 ]     (* W19, ENP *)
  // as ST:
  //   IF ENP <= VNM THEN W19 := ENP; END_IF;

// Rung 60
  LD [ %MF28 > %MF85 ]    (* ENP, VNM *)
  [ %MF235 := %MF85 ]     (* W19, VNM *)
  // as ST:
  //   IF ENP > VNM THEN W19 := VNM; END_IF;

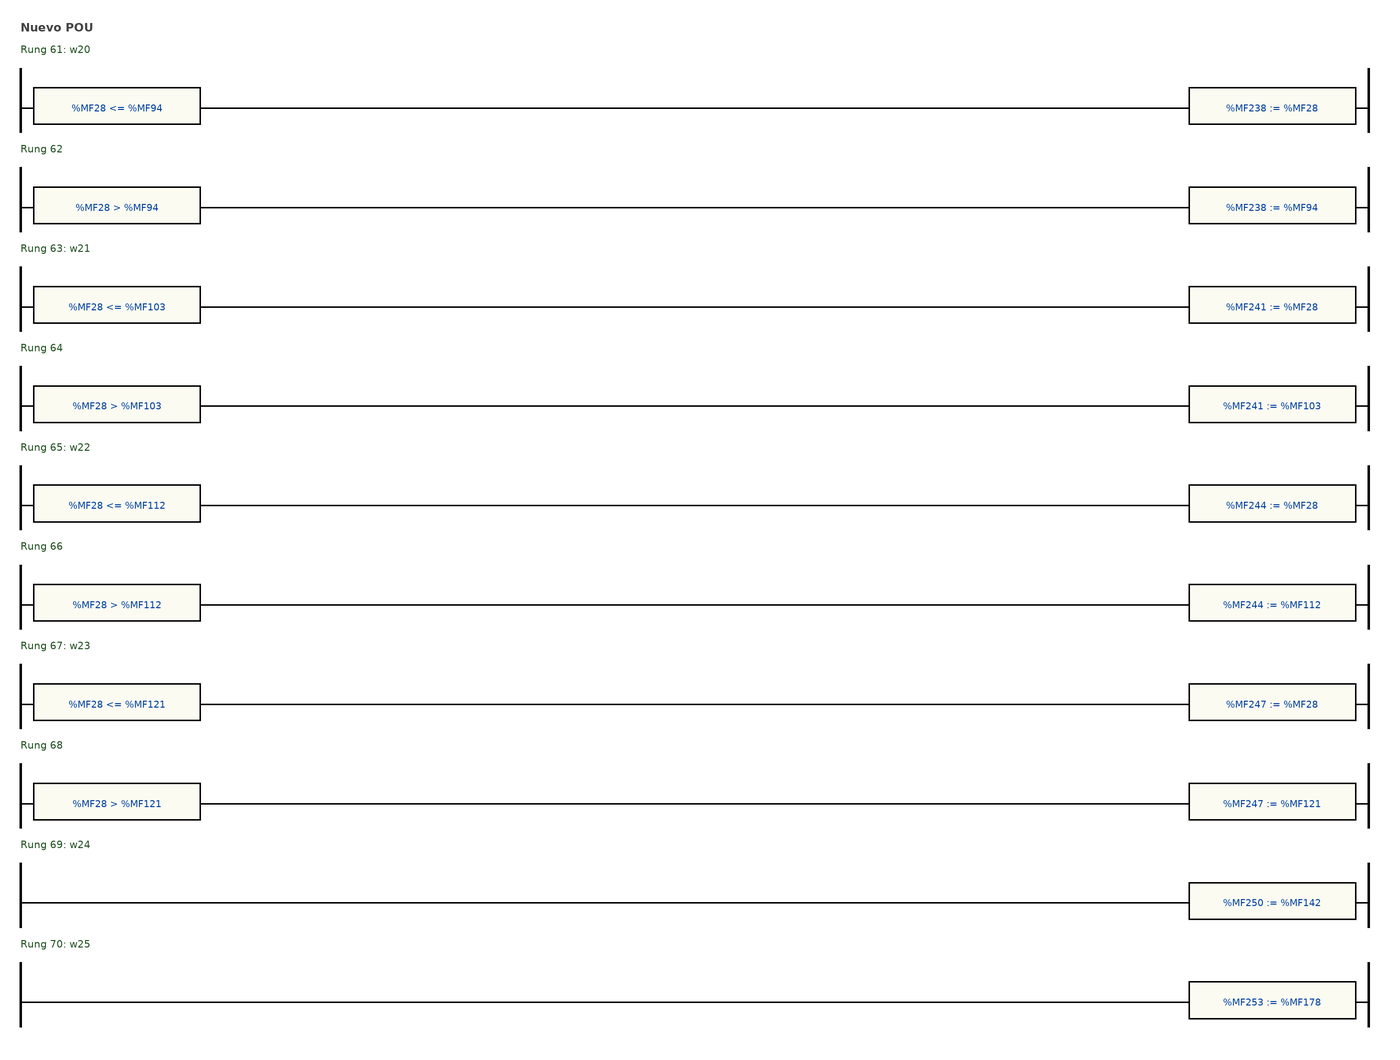

// Rung 61: w20
  LD [ %MF28 <= %MF94 ]   (* ENP, VNP *)
  [ %MF238 := %MF28 ]     (* W20, ENP *)
  // as ST:
  //   IF ENP <= VNP THEN W20 := ENP; END_IF;

// Rung 62
  LD [ %MF28 > %MF94 ]    (* ENP, VNP *)
  [ %MF238 := %MF94 ]     (* W20, VNP *)
  // as ST:
  //   IF ENP > VNP THEN W20 := VNP; END_IF;

// Rung 63: w21
  LD [ %MF28 <= %MF103 ]  (* ENP, VZ *)
  [ %MF241 := %MF28 ]     (* W21, ENP *)
  // as ST:
  //   IF ENP <= VZ THEN W21 := ENP; END_IF;

// Rung 64
  LD [ %MF28 > %MF103 ]   (* ENP, VZ *)
  [ %MF241 := %MF103 ]    (* W21, VZ *)
  // as ST:
  //   IF ENP > VZ THEN W21 := VZ; END_IF;

// Rung 65: w22
  LD [ %MF28 <= %MF112 ]  (* ENP, VPP *)
  [ %MF244 := %MF28 ]     (* W22, ENP *)
  // as ST:
  //   IF ENP <= VPP THEN W22 := ENP; END_IF;

// Rung 66
  LD [ %MF28 > %MF112 ]   (* ENP, VPP *)
  [ %MF244 := %MF112 ]    (* W22, VPP *)
  // as ST:
  //   IF ENP > VPP THEN W22 := VPP; END_IF;

// Rung 67: w23
  LD [ %MF28 <= %MF121 ]  (* ENP, VPM *)
  [ %MF247 := %MF28 ]     (* W23, ENP *)
  // as ST:
  //   IF ENP <= VPM THEN W23 := ENP; END_IF;

// Rung 68
  LD [ %MF28 > %MF121 ]   (* ENP, VPM *)
  [ %MF247 := %MF121 ]    (* W23, VPM *)
  // as ST:
  //   IF ENP > VPM THEN W23 := VPM; END_IF;

// Rung 69: w24
  LD 1
  [ %MF250 := %MF142 ]    (* W24, NL *)
  // as ST:
  //   W24 := NL;

// Rung 70: w25
  LD 1
  [ %MF253 := %MF178 ]    (* W25, PL *)
  // as ST:
  //   W25 := PL;

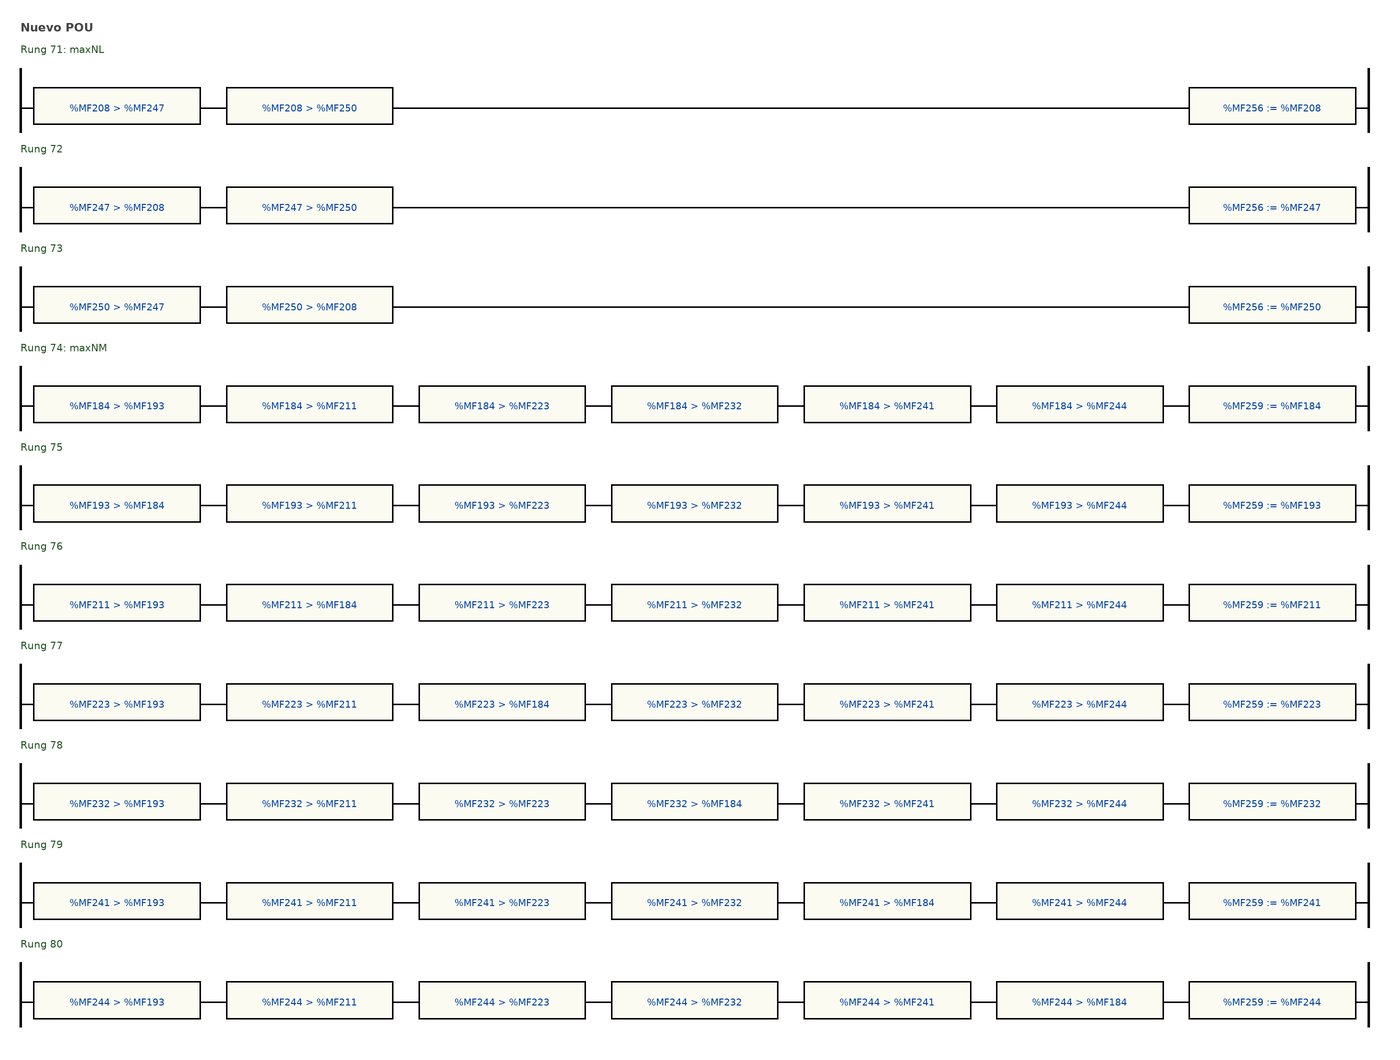

// Rung 71: maxNL
  LD [ %MF208 > %MF247 ]  (* W10, W23 *)
  AND [ %MF208 > %MF250 ] (* W10, W24 *)
  [ %MF256 := %MF208 ]    (* U_NL, W10 *)
  // as ST:
  //   IF W10 > W23 AND W10 > W24 THEN U_NL := W10; END_IF;

// Rung 72
  LD [ %MF247 > %MF208 ]  (* W23, W10 *)
  AND [ %MF247 > %MF250 ] (* W23, W24 *)
  [ %MF256 := %MF247 ]    (* U_NL, W23 *)
  // as ST:
  //   IF W23 > W10 AND W23 > W24 THEN U_NL := W23; END_IF;

// Rung 73
  LD [ %MF250 > %MF247 ]  (* W24, W23 *)
  AND [ %MF250 > %MF208 ] (* W24, W10 *)
  [ %MF256 := %MF250 ]    (* U_NL, W24 *)
  // as ST:
  //   IF W24 > W23 AND W24 > W10 THEN U_NL := W24; END_IF;

// Rung 74: maxNM
  LD [ %MF184 > %MF193 ]  (* W2, W5 *)
  AND [ %MF184 > %MF211 ] (* W2, W11 *)
  AND [ %MF184 > %MF223 ] (* W2, W15 *)
  AND [ %MF184 > %MF232 ] (* W2, W18 *)
  AND [ %MF184 > %MF241 ] (* W2, W21 *)
  AND [ %MF184 > %MF244 ] (* W2, W22 *)
  [ %MF259 := %MF184 ]    (* U_NM, W2 *)
  // as ST:
  //   IF W2 > W5 AND W2 > W11 AND W2 > W15 AND W2 > W18 AND W2 > W21 AND W2 > W22 THEN U_NM := W2; END_IF;

// Rung 75
  LD [ %MF193 > %MF184 ]  (* W5, W2 *)
  AND [ %MF193 > %MF211 ] (* W5, W11 *)
  AND [ %MF193 > %MF223 ] (* W5, W15 *)
  AND [ %MF193 > %MF232 ] (* W5, W18 *)
  AND [ %MF193 > %MF241 ] (* W5, W21 *)
  AND [ %MF193 > %MF244 ] (* W5, W22 *)
  [ %MF259 := %MF193 ]    (* U_NM, W5 *)
  // as ST:
  //   IF W5 > W2 AND W5 > W11 AND W5 > W15 AND W5 > W18 AND W5 > W21 AND W5 > W22 THEN U_NM := W5; END_IF;

// Rung 76
  LD [ %MF211 > %MF193 ]  (* W11, W5 *)
  AND [ %MF211 > %MF184 ] (* W11, W2 *)
  AND [ %MF211 > %MF223 ] (* W11, W15 *)
  AND [ %MF211 > %MF232 ] (* W11, W18 *)
  AND [ %MF211 > %MF241 ] (* W11, W21 *)
  AND [ %MF211 > %MF244 ] (* W11, W22 *)
  [ %MF259 := %MF211 ]    (* U_NM, W11 *)
  // as ST:
  //   IF W11 > W5 AND W11 > W2 AND W11 > W15 AND W11 > W18 AND W11 > W21 AND W11 > W22 THEN U_NM := W11; END_IF;

// Rung 77
  LD [ %MF223 > %MF193 ]  (* W15, W5 *)
  AND [ %MF223 > %MF211 ] (* W15, W11 *)
  AND [ %MF223 > %MF184 ] (* W15, W2 *)
  AND [ %MF223 > %MF232 ] (* W15, W18 *)
  AND [ %MF223 > %MF241 ] (* W15, W21 *)
  AND [ %MF223 > %MF244 ] (* W15, W22 *)
  [ %MF259 := %MF223 ]    (* U_NM, W15 *)
  // as ST:
  //   IF W15 > W5 AND W15 > W11 AND W15 > W2 AND W15 > W18 AND W15 > W21 AND W15 > W22 THEN U_NM := W15; END_IF;

// Rung 78
  LD [ %MF232 > %MF193 ]  (* W18, W5 *)
  AND [ %MF232 > %MF211 ] (* W18, W11 *)
  AND [ %MF232 > %MF223 ] (* W18, W15 *)
  AND [ %MF232 > %MF184 ] (* W18, W2 *)
  AND [ %MF232 > %MF241 ] (* W18, W21 *)
  AND [ %MF232 > %MF244 ] (* W18, W22 *)
  [ %MF259 := %MF232 ]    (* U_NM, W18 *)
  // as ST:
  //   IF W18 > W5 AND W18 > W11 AND W18 > W15 AND W18 > W2 AND W18 > W21 AND W18 > W22 THEN U_NM := W18; END_IF;

// Rung 79
  LD [ %MF241 > %MF193 ]  (* W21, W5 *)
  AND [ %MF241 > %MF211 ] (* W21, W11 *)
  AND [ %MF241 > %MF223 ] (* W21, W15 *)
  AND [ %MF241 > %MF232 ] (* W21, W18 *)
  AND [ %MF241 > %MF184 ] (* W21, W2 *)
  AND [ %MF241 > %MF244 ] (* W21, W22 *)
  [ %MF259 := %MF241 ]    (* U_NM, W21 *)
  // as ST:
  //   IF W21 > W5 AND W21 > W11 AND W21 > W15 AND W21 > W18 AND W21 > W2 AND W21 > W22 THEN U_NM := W21; END_IF;

// Rung 80
  LD [ %MF244 > %MF193 ]  (* W22, W5 *)
  AND [ %MF244 > %MF211 ] (* W22, W11 *)
  AND [ %MF244 > %MF223 ] (* W22, W15 *)
  AND [ %MF244 > %MF232 ] (* W22, W18 *)
  AND [ %MF244 > %MF241 ] (* W22, W21 *)
  AND [ %MF244 > %MF184 ] (* W22, W2 *)
  [ %MF259 := %MF244 ]    (* U_NM, W22 *)
  // as ST:
  //   IF W22 > W5 AND W22 > W11 AND W22 > W15 AND W22 > W18 AND W22 > W21 AND W22 > W2 THEN U_NM := W22; END_IF;

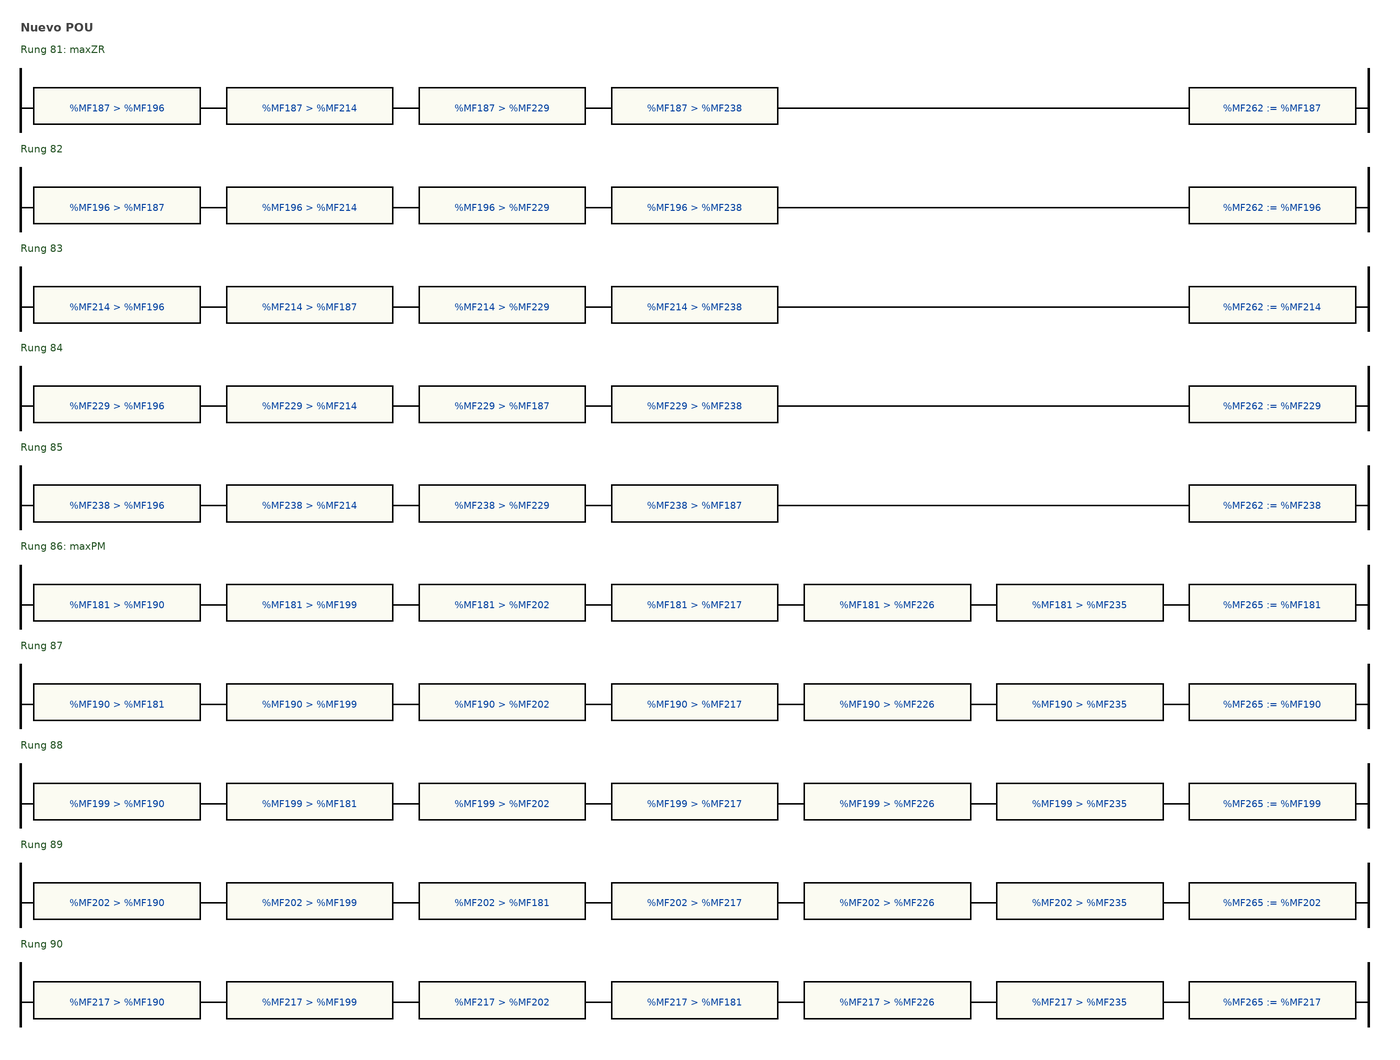

// Rung 81: maxZR
  LD [ %MF187 > %MF196 ]  (* W3, W6 *)
  AND [ %MF187 > %MF214 ] (* W3, W12 *)
  AND [ %MF187 > %MF229 ] (* W3, W17 *)
  AND [ %MF187 > %MF238 ] (* W3, W20 *)
  [ %MF262 := %MF187 ]    (* U_ZR, W3 *)
  // as ST:
  //   IF W3 > W6 AND W3 > W12 AND W3 > W17 AND W3 > W20 THEN U_ZR := W3; END_IF;

// Rung 82
  LD [ %MF196 > %MF187 ]  (* W6, W3 *)
  AND [ %MF196 > %MF214 ] (* W6, W12 *)
  AND [ %MF196 > %MF229 ] (* W6, W17 *)
  AND [ %MF196 > %MF238 ] (* W6, W20 *)
  [ %MF262 := %MF196 ]    (* U_ZR, W6 *)
  // as ST:
  //   IF W6 > W3 AND W6 > W12 AND W6 > W17 AND W6 > W20 THEN U_ZR := W6; END_IF;

// Rung 83
  LD [ %MF214 > %MF196 ]  (* W12, W6 *)
  AND [ %MF214 > %MF187 ] (* W12, W3 *)
  AND [ %MF214 > %MF229 ] (* W12, W17 *)
  AND [ %MF214 > %MF238 ] (* W12, W20 *)
  [ %MF262 := %MF214 ]    (* U_ZR, W12 *)
  // as ST:
  //   IF W12 > W6 AND W12 > W3 AND W12 > W17 AND W12 > W20 THEN U_ZR := W12; END_IF;

// Rung 84
  LD [ %MF229 > %MF196 ]  (* W17, W6 *)
  AND [ %MF229 > %MF214 ] (* W17, W12 *)
  AND [ %MF229 > %MF187 ] (* W17, W3 *)
  AND [ %MF229 > %MF238 ] (* W17, W20 *)
  [ %MF262 := %MF229 ]    (* U_ZR, W17 *)
  // as ST:
  //   IF W17 > W6 AND W17 > W12 AND W17 > W3 AND W17 > W20 THEN U_ZR := W17; END_IF;

// Rung 85
  LD [ %MF238 > %MF196 ]  (* W20, W6 *)
  AND [ %MF238 > %MF214 ] (* W20, W12 *)
  AND [ %MF238 > %MF229 ] (* W20, W17 *)
  AND [ %MF238 > %MF187 ] (* W20, W3 *)
  [ %MF262 := %MF238 ]    (* U_ZR, W20 *)
  // as ST:
  //   IF W20 > W6 AND W20 > W12 AND W20 > W17 AND W20 > W3 THEN U_ZR := W20; END_IF;

// Rung 86: maxPM
  LD [ %MF181 > %MF190 ]  (* W1, W4 *)
  AND [ %MF181 > %MF199 ] (* W1, W7 *)
  AND [ %MF181 > %MF202 ] (* W1, W8 *)
  AND [ %MF181 > %MF217 ] (* W1, W13 *)
  AND [ %MF181 > %MF226 ] (* W1, W16 *)
  AND [ %MF181 > %MF235 ] (* W1, W19 *)
  [ %MF265 := %MF181 ]    (* U_PM, W1 *)
  // as ST:
  //   IF W1 > W4 AND W1 > W7 AND W1 > W8 AND W1 > W13 AND W1 > W16 AND W1 > W19 THEN U_PM := W1; END_IF;

// Rung 87
  LD [ %MF190 > %MF181 ]  (* W4, W1 *)
  AND [ %MF190 > %MF199 ] (* W4, W7 *)
  AND [ %MF190 > %MF202 ] (* W4, W8 *)
  AND [ %MF190 > %MF217 ] (* W4, W13 *)
  AND [ %MF190 > %MF226 ] (* W4, W16 *)
  AND [ %MF190 > %MF235 ] (* W4, W19 *)
  [ %MF265 := %MF190 ]    (* U_PM, W4 *)
  // as ST:
  //   IF W4 > W1 AND W4 > W7 AND W4 > W8 AND W4 > W13 AND W4 > W16 AND W4 > W19 THEN U_PM := W4; END_IF;

// Rung 88
  LD [ %MF199 > %MF190 ]  (* W7, W4 *)
  AND [ %MF199 > %MF181 ] (* W7, W1 *)
  AND [ %MF199 > %MF202 ] (* W7, W8 *)
  AND [ %MF199 > %MF217 ] (* W7, W13 *)
  AND [ %MF199 > %MF226 ] (* W7, W16 *)
  AND [ %MF199 > %MF235 ] (* W7, W19 *)
  [ %MF265 := %MF199 ]    (* U_PM, W7 *)
  // as ST:
  //   IF W7 > W4 AND W7 > W1 AND W7 > W8 AND W7 > W13 AND W7 > W16 AND W7 > W19 THEN U_PM := W7; END_IF;

// Rung 89
  LD [ %MF202 > %MF190 ]  (* W8, W4 *)
  AND [ %MF202 > %MF199 ] (* W8, W7 *)
  AND [ %MF202 > %MF181 ] (* W8, W1 *)
  AND [ %MF202 > %MF217 ] (* W8, W13 *)
  AND [ %MF202 > %MF226 ] (* W8, W16 *)
  AND [ %MF202 > %MF235 ] (* W8, W19 *)
  [ %MF265 := %MF202 ]    (* U_PM, W8 *)
  // as ST:
  //   IF W8 > W4 AND W8 > W7 AND W8 > W1 AND W8 > W13 AND W8 > W16 AND W8 > W19 THEN U_PM := W8; END_IF;

// Rung 90
  LD [ %MF217 > %MF190 ]  (* W13, W4 *)
  AND [ %MF217 > %MF199 ] (* W13, W7 *)
  AND [ %MF217 > %MF202 ] (* W13, W8 *)
  AND [ %MF217 > %MF181 ] (* W13, W1 *)
  AND [ %MF217 > %MF226 ] (* W13, W16 *)
  AND [ %MF217 > %MF235 ] (* W13, W19 *)
  [ %MF265 := %MF217 ]    (* U_PM, W13 *)
  // as ST:
  //   IF W13 > W4 AND W13 > W7 AND W13 > W8 AND W13 > W1 AND W13 > W16 AND W13 > W19 THEN U_PM := W13; END_IF;

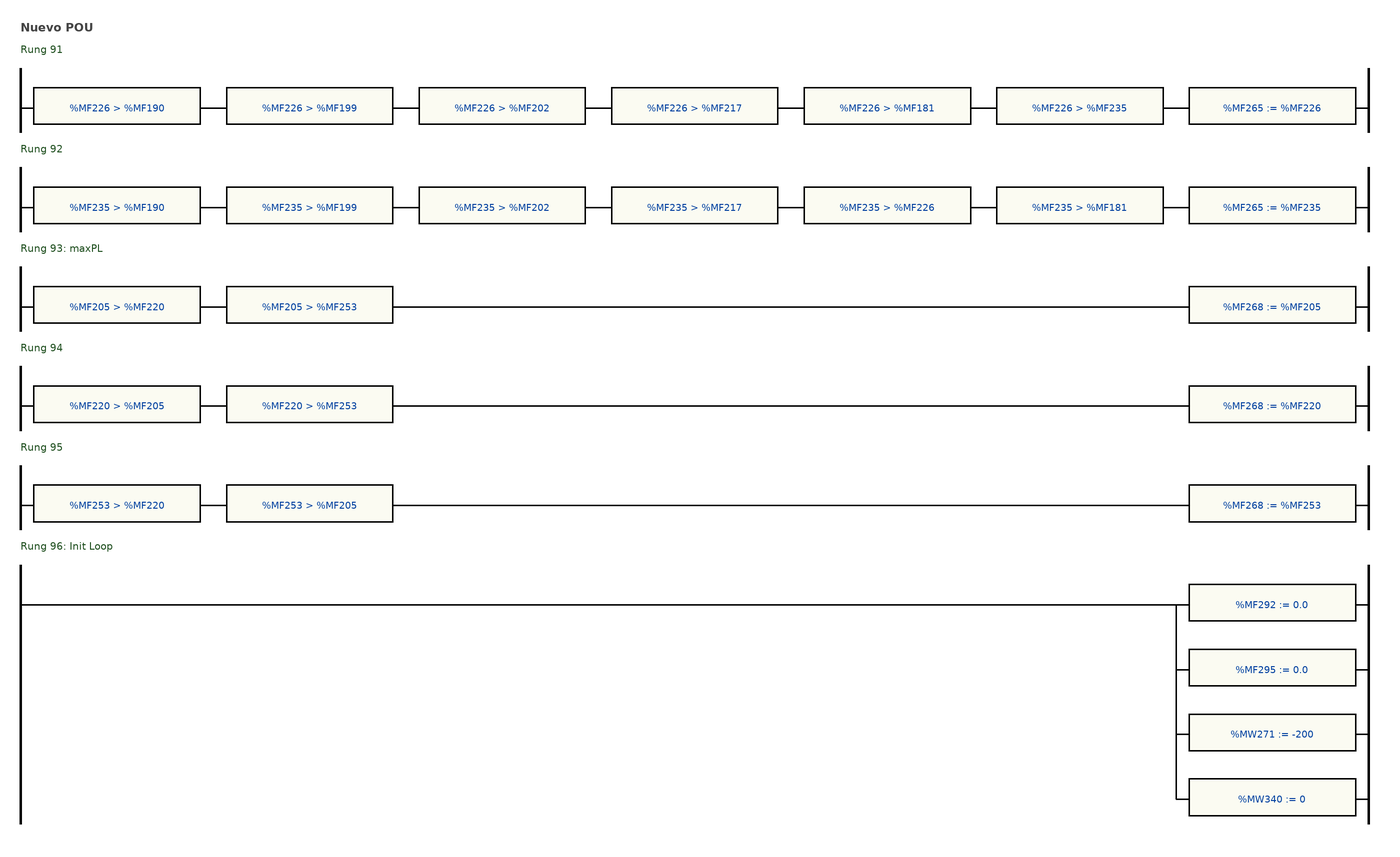

// Rung 91
  LD [ %MF226 > %MF190 ]  (* W16, W4 *)
  AND [ %MF226 > %MF199 ] (* W16, W7 *)
  AND [ %MF226 > %MF202 ] (* W16, W8 *)
  AND [ %MF226 > %MF217 ] (* W16, W13 *)
  AND [ %MF226 > %MF181 ] (* W16, W1 *)
  AND [ %MF226 > %MF235 ] (* W16, W19 *)
  [ %MF265 := %MF226 ]    (* U_PM, W16 *)
  // as ST:
  //   IF W16 > W4 AND W16 > W7 AND W16 > W8 AND W16 > W13 AND W16 > W1 AND W16 > W19 THEN U_PM := W16; END_IF;

// Rung 92
  LD [ %MF235 > %MF190 ]  (* W19, W4 *)
  AND [ %MF235 > %MF199 ] (* W19, W7 *)
  AND [ %MF235 > %MF202 ] (* W19, W8 *)
  AND [ %MF235 > %MF217 ] (* W19, W13 *)
  AND [ %MF235 > %MF226 ] (* W19, W16 *)
  AND [ %MF235 > %MF181 ] (* W19, W1 *)
  [ %MF265 := %MF235 ]    (* U_PM, W19 *)
  // as ST:
  //   IF W19 > W4 AND W19 > W7 AND W19 > W8 AND W19 > W13 AND W19 > W16 AND W19 > W1 THEN U_PM := W19; END_IF;

// Rung 93: maxPL
  LD [ %MF205 > %MF220 ]  (* W9, W14 *)
  AND [ %MF205 > %MF253 ] (* W9, W25 *)
  [ %MF268 := %MF205 ]    (* U_PL, W9 *)
  // as ST:
  //   IF W9 > W14 AND W9 > W25 THEN U_PL := W9; END_IF;

// Rung 94
  LD [ %MF220 > %MF205 ]  (* W14, W9 *)
  AND [ %MF220 > %MF253 ] (* W14, W25 *)
  [ %MF268 := %MF220 ]    (* U_PL, W14 *)
  // as ST:
  //   IF W14 > W9 AND W14 > W25 THEN U_PL := W14; END_IF;

// Rung 95
  LD [ %MF253 > %MF220 ]  (* W25, W14 *)
  AND [ %MF253 > %MF205 ] (* W25, W9 *)
  [ %MF268 := %MF253 ]    (* U_PL, W25 *)
  // as ST:
  //   IF W25 > W14 AND W25 > W9 THEN U_PL := W25; END_IF;

// Rung 96: Init Loop
  LD 1
  [ %MF292 := 0.0 ]
  [ %MF295 := 0.0 ]
  [ %MW271 := -200 ]      (* CONT *)
  [ %MW340 := 0 ]
  // as ST:
  //   %MF292 := 0.0;
  //   %MF295 := 0.0;
  //   CONT := -200;
  //   %MW340 := 0;

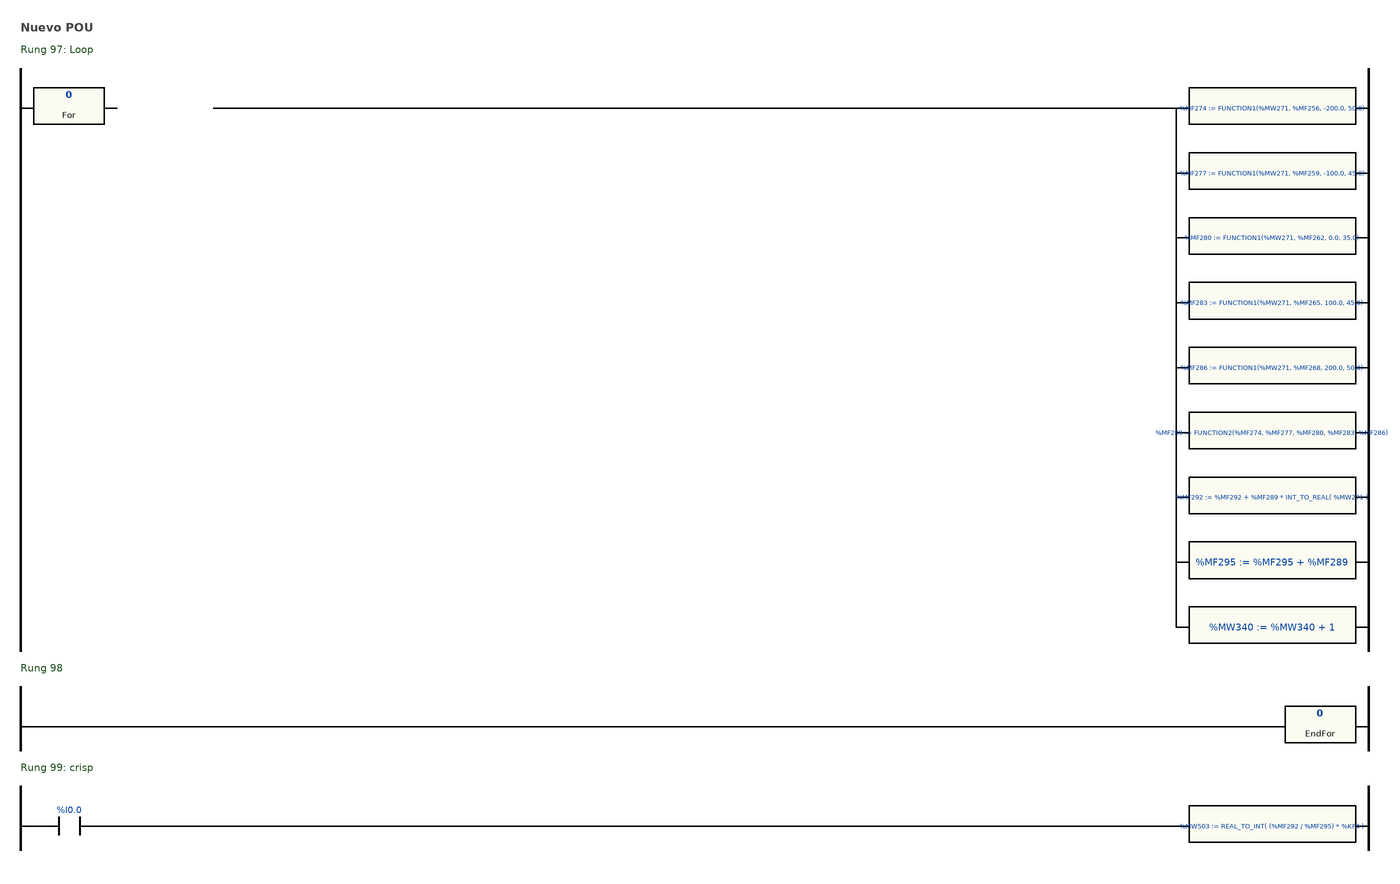

// Rung 97: Loop
  FOR0 ( %MW271 , %MW271 , <= , 200 , 4 )(* CONT, CONT *)
  [ %MF274 := FUNCTION1 ( %MW271 , %MF256 , -200.0 , 50.0 ) ](* CONT, U_NL *)
  [ %MF277 := FUNCTION1 ( %MW271 , %MF259 , -100.0 , 45.0 ) ](* CONT, U_NM *)
  [ %MF280 := FUNCTION1 ( %MW271 , %MF262 , 0.0 , 35.0 ) ](* CONT, U_ZR *)
  [ %MF283 := FUNCTION1 ( %MW271 , %MF265 , 100.0 , 45.0 ) ](* CONT, U_PM *)
  [ %MF286 := FUNCTION1 ( %MW271 , %MF268 , 200.0 , 50.0 ) ](* CONT, U_PL *)
  [ %MF289 := FUNCTION2 ( %MF274 , %MF277 , %MF280 , %MF283 , %MF286 ) ]
  [ %MF292 := %MF292 + %MF289 * INT_TO_REAL ( %MW271 ) ](* CONT *)
  [ %MF295 := %MF295 + %MF289 ]
  [ %MW340 := %MW340 + 1 ]

// Rung 98
  LD 1
  ENDFOR0

// Rung 99: crisp
  LD %I0.0
  [ %MW503 := REAL_TO_INT ( ( %MF292 / %MF295 ) * %KF4 ) ](* CRISP, CONV_OUTPUT *)
  // as ST:
  //   IF %I0.0 THEN CRISP := REAL_TO_INT ( ( %MF292 / %MF295 ) * CONV_OUTPUT ); END_IF;

UserFunctionPou FUNCTION1
  (* SectionNumber=2 *)

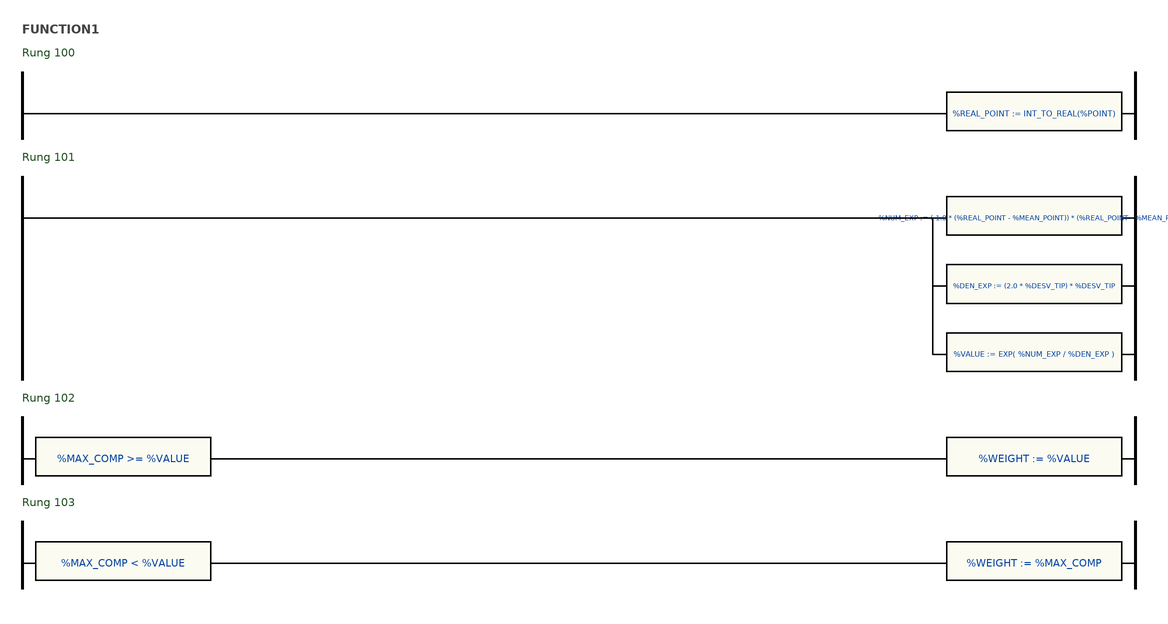

// Rung 100
  LD 1
  [ %REAL_POINT := INT_TO_REAL ( %POINT ) ]
  // as ST:
  //   %REAL_POINT := INT_TO_REAL ( %POINT );

// Rung 101
  LD 1
  [ %NUM_EXP := ( -1.0 * ( %REAL_POINT - %MEAN_POINT ) ) * ( %REAL_POINT - %MEAN_POINT ) ]
  [ %DEN_EXP := ( 2.0 * %DESV_TIP ) * %DESV_TIP ]
  [ %VALUE := EXP ( %NUM_EXP / %DEN_EXP ) ]
  // as ST:
  //   %NUM_EXP := ( -1.0 * ( %REAL_POINT - %MEAN_POINT ) ) * ( %REAL_POINT - %MEAN_POINT );
  //   %DEN_EXP := ( 2.0 * %DESV_TIP ) * %DESV_TIP;
  //   %VALUE := EXP ( %NUM_EXP / %DEN_EXP );

// Rung 102
  LD [ %MAX_COMP >= %VALUE ]
  [ %WEIGHT := %VALUE ]
  // as ST:
  //   IF %MAX_COMP >= %VALUE THEN %WEIGHT := %VALUE; END_IF;

// Rung 103
  LD [ %MAX_COMP < %VALUE ]
  [ %WEIGHT := %MAX_COMP ]
  // as ST:
  //   IF %MAX_COMP < %VALUE THEN %WEIGHT := %MAX_COMP; END_IF;

UserFunctionPou FUNCTION2
  (* SectionNumber=3 *)

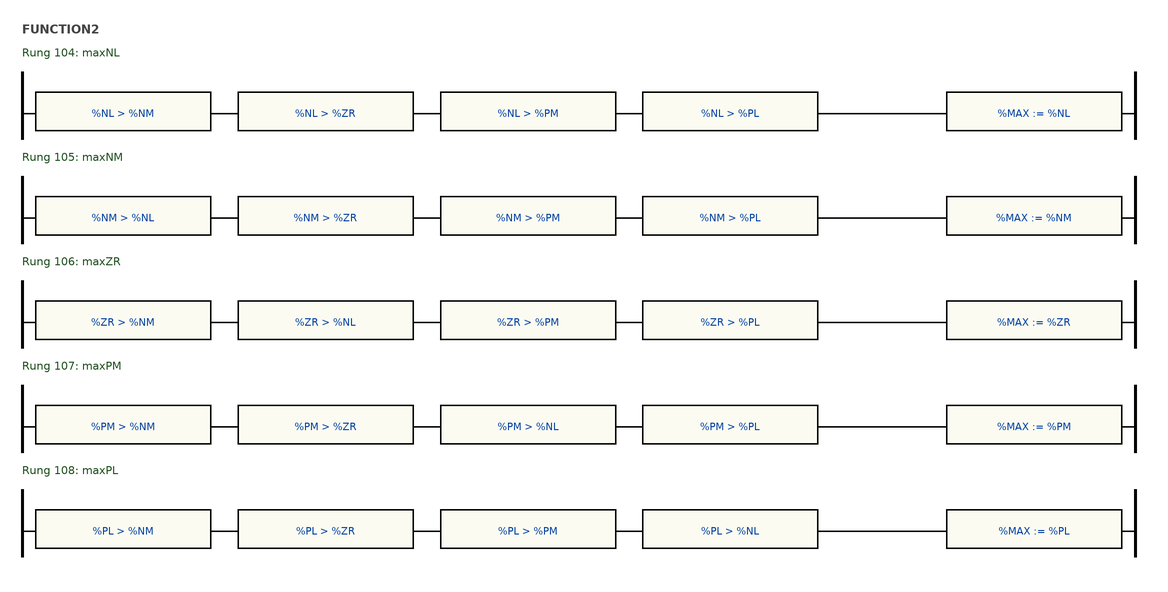

// Rung 104: maxNL
  LD [ %NL > %NM ]
  AND [ %NL > %ZR ]
  AND [ %NL > %PM ]
  AND [ %NL > %PL ]
  [ %MAX := %NL ]
  // as ST:
  //   IF %NL > %NM AND %NL > %ZR AND %NL > %PM AND %NL > %PL THEN %MAX := %NL; END_IF;

// Rung 105: maxNM
  LD [ %NM > %NL ]
  AND [ %NM > %ZR ]
  AND [ %NM > %PM ]
  AND [ %NM > %PL ]
  [ %MAX := %NM ]
  // as ST:
  //   IF %NM > %NL AND %NM > %ZR AND %NM > %PM AND %NM > %PL THEN %MAX := %NM; END_IF;

// Rung 106: maxZR
  LD [ %ZR > %NM ]
  AND [ %ZR > %NL ]
  AND [ %ZR > %PM ]
  AND [ %ZR > %PL ]
  [ %MAX := %ZR ]
  // as ST:
  //   IF %ZR > %NM AND %ZR > %NL AND %ZR > %PM AND %ZR > %PL THEN %MAX := %ZR; END_IF;

// Rung 107: maxPM
  LD [ %PM > %NM ]
  AND [ %PM > %ZR ]
  AND [ %PM > %NL ]
  AND [ %PM > %PL ]
  [ %MAX := %PM ]
  // as ST:
  //   IF %PM > %NM AND %PM > %ZR AND %PM > %NL AND %PM > %PL THEN %MAX := %PM; END_IF;

// Rung 108: maxPL
  LD [ %PL > %NM ]
  AND [ %PL > %ZR ]
  AND [ %PL > %PM ]
  AND [ %PL > %NL ]
  [ %MAX := %PL ]
  // as ST:
  //   IF %PL > %NM AND %PL > %ZR AND %PL > %PM AND %PL > %NL THEN %MAX := %PL; END_IF;
